LIN {X 0,Y 284.193,Z 792.338,A -85,B 0,C 180,E1 16435.65,E2 16435.65} C_VEL
LIN {X 0,Y 275.5,Z 813.457,A -85,B 0,C 180,E1 16443.138,E2 16443.138} C_VEL
LIN {X 0,Y 270.881,Z 827.883,A -85,B 0,C 180,E1 16450.476,E2 16450.476} C_VEL
LIN {X 0,Y 268.896,Z 838.261,A -85,B 0,C 180,E1 16458.673,E2 16458.673} C_VEL
LIN {X 0,Y 268.674,Z 843.154,A -85,B 0,C 180,E1 16466.783,E2 16466.783} C_VEL
LIN {X 0,Y 269.021,Z 843.604,A -85,B 0,C 180,E1 16470.002,E2 16470.002} C_VEL
LIN {X 0,Y 268.664,Z 840.876,A -85,B 0,C 180,E1 16478.074,E2 16478.074} C_VEL
LIN {X 0,Y 269.781,Z 832.628,A -85,B 0,C 180,E1 16486.243,E2 16486.243} C_VEL
LIN {X 0,Y 273.657,Z 818.429,A -85,B 0,C 180,E1 16494.453,E2 16494.453} C_VEL
LIN {X 0,Y 281.012,Z 798.576,A -85,B 0,C 180,E1 16502.079,E2 16502.079} C_VEL
LIN {X 0,Y 291.199,Z 773.618,A -85,B 0,C 180,E1 16508.743,E2 16508.743} C_VEL
LIN {X 0,Y 302.271,Z 746.073,A -85,B 0,C 180,E1 16513.948,E2 16513.948} C_VEL
LIN {X 0,Y 314,Z 714.004,A -85,B 0,C 180,E1 16518.227,E2 16518.227} C_VEL
LIN {X 0,Y 324.739,Z 678.752,A -85,B 0,C 180,E1 16521.486,E2 16521.486} C_VEL
LIN {X 0,Y 328.308,Z 663.259,A -85,B 0,C 180,E1 16522.637,E2 16522.637} C_VEL
LIN {X 0,Y 318.026,Z 633.867,A -85,B 0,C 180,E1 16527.518,E2 16527.518} C_VEL
LIN {X 0,Y 305.742,Z 608.81,A -85,B 0,C 180,E1 16532.476,E2 16532.476} C_VEL
LIN {X 0,Y 298.214,Z 601.214,A -85,B 0,C 180,E1 16535.1,E2 16535.1} C_VEL
LIN {X 0,Y 290.45,Z 594.981,A -85,B 0,C 180,E1 16537.97,E2 16537.97} C_VEL
LIN {X 0,Y 278.094,Z 576.688,A -85,B 0,C 180,E1 16543.729,E2 16543.729} C_VEL
LIN {X 0,Y 272.613,Z 569.407,A -85,B 0,C 180,E1 16546.675,E2 16546.675} C_VEL
LIN {X 0,Y 268.838,Z 563.675,A -85,B 0,C 180,E1 16549.01,E2 16549.01} C_VEL
LIN {X 0,Y 265.24,Z 558.237,A -85,B 0,C 180,E1 16551.479,E2 16551.479} C_VEL
LIN {X 0,Y 260.078,Z 551.896,A -85,B 0,C 180,E1 16555.502,E2 16555.502} C_VEL
LIN {X 0,Y 259.824,Z 549.53,A -85,B 0,C 180,E1 16556.227,E2 16556.227} C_VEL
LIN {X 0,Y 260.166,Z 549.53,A -85,B 0,C 180,E1 16559.972,E2 16559.972} C_VEL
LIN {X 0,Y 259.366,Z 549.53,A -85,B 0,C 180,E1 16568.461,E2 16568.461} C_VEL
LIN {X 0,Y 258.757,Z 549.53,A -85,B 0,C 180,E1 16576.92,E2 16576.92} C_VEL
LIN {X 0,Y 258.263,Z 549.53,A -85,B 0,C 180,E1 16584.106,E2 16584.106} C_VEL
LIN {X 0,Y 257.894,Z 549.53,A -85,B 0,C 180,E1 16591.736,E2 16591.736} C_VEL
LIN {X 0,Y 257.813,Z 549.77,A -85,B 0,C 180,E1 16595.549,E2 16595.549} C_VEL
LIN {X 0,Y 259.44,Z 554.315,A -85,B 0,C 180,E1 16597.326,E2 16597.326} C_VEL
LIN {X 0,Y 263.605,Z 557.866,A -85,B 0,C 180,E1 16600.498,E2 16600.498} C_VEL
LIN {X 0,Y 267.187,Z 563.441,A -85,B 0,C 180,E1 16603.061,E2 16603.061} C_VEL
LIN {X 0,Y 269.471,Z 566.342,A -85,B 0,C 180,E1 16604.516,E2 16604.516} C_VEL
LIN {X 0,Y 279.761,Z 580.464,A -85,B 0,C 180,E1 16610.268,E2 16610.268} C_VEL
LIN {X 0,Y 291.304,Z 599.056,A -85,B 0,C 180,E1 16616.073,E2 16616.073} C_VEL
LIN {X 0,Y 302.413,Z 621.809,A -85,B 0,C 180,E1 16621.67,E2 16621.67} C_VEL
LIN {X 0,Y 310.963,Z 646.908,A -85,B 0,C 180,E1 16626.849,E2 16626.849} C_VEL
LIN {X 0,Y 313.377,Z 660.612,A -85,B 0,C 180,E1 16629.324,E2 16629.324} C_VEL
LIN {X 0,Y 302.378,Z 694.403,A -85,B 0,C 180,E1 16633.136,E2 16633.136} C_VEL
LIN {X 0,Y 290.875,Z 723.87,A -85,B 0,C 180,E1 16638.021,E2 16638.021} C_VEL
LIN {X 0,Y 280.218,Z 748.211,A -85,B 0,C 180,E1 16643.815,E2 16643.815} C_VEL
LIN {X 0,Y 271.445,Z 767.751,A -85,B 0,C 180,E1 16650.553,E2 16650.553} C_VEL
LIN {X 0,Y 265.654,Z 781.533,A -85,B 0,C 180,E1 16657.597,E2 16657.597} C_VEL
LIN {X 0,Y 262.351,Z 790.678,A -85,B 0,C 180,E1 16664.998,E2 16664.998} C_VEL
LIN {X 0,Y 260.523,Z 795.27,A -85,B 0,C 180,E1 16672.171,E2 16672.171} C_VEL
LIN {X 0,Y 260.569,Z 795.838,A -85,B 0,C 180,E1 16679.773,E2 16679.773} C_VEL
LIN {X 0,Y 262.859,Z 791.758,A -85,B 0,C 180,E1 16687.666,E2 16687.666} C_VEL
LIN {X 0,Y 267.17,Z 782.441,A -85,B 0,C 180,E1 16695.737,E2 16695.737} C_VEL
LIN {X 0,Y 274.41,Z 768.233,A -85,B 0,C 180,E1 16703.143,E2 16703.143} C_VEL
LIN {X 0,Y 284.656,Z 748.679,A -85,B 0,C 180,E1 16709.894,E2 16709.894} C_VEL
LIN {X 0,Y 297.561,Z 722.75,A -85,B 0,C 180,E1 16715.894,E2 16715.894} C_VEL
LIN {X 0,Y 310.18,Z 693.863,A -85,B 0,C 180,E1 16720.466,E2 16720.466} C_VEL
LIN {X 0,Y 320.732,Z 664.253,A -85,B 0,C 180,E1 16723.806,E2 16723.806} C_VEL
LIN {X 0,Y 317.188,Z 642.293,A -85,B 0,C 180,E1 16728.708,E2 16728.708} C_VEL
LIN {X 0,Y 312.027,Z 624.584,A -85,B 0,C 180,E1 16733.778,E2 16733.778} C_VEL
LIN {X 0,Y 307.138,Z 612.298,A -85,B 0,C 180,E1 16738.842,E2 16738.842} C_VEL
LIN {X 0,Y 304.838,Z 607,A -85,B 0,C 180,E1 16741.993,E2 16741.993} C_VEL
LIN {X 0,Y 303.417,Z 603.216,A -85,B 0,C 180,E1 16744.94,E2 16744.94} C_VEL
LIN {X 0,Y 303.196,Z 603.27,A -85,B 0,C 180,E1 16754.063,E2 16754.063} C_VEL
LIN {X 0,Y 307.12,Z 611.288,A -85,B 0,C 180,E1 16760.137,E2 16760.137} C_VEL
LIN {X 0,Y 312.817,Z 623.081,A -85,B 0,C 180,E1 16765.242,E2 16765.242} C_VEL
LIN {X 0,Y 320.158,Z 641.035,A -85,B 0,C 180,E1 16770.477,E2 16770.477} C_VEL
LIN {X 0,Y 326.227,Z 663.874,A -85,B 0,C 180,E1 16775.218,E2 16775.218} C_VEL
LIN {X 0,Y 326.696,Z 668.857,A -85,B 0,C 180,E1 16775.992,E2 16775.992} C_VEL
LIN {X 0,Y 314.613,Z 705.853,A -85,B 0,C 180,E1 16779.162,E2 16779.162} C_VEL
LIN {X 0,Y 301.662,Z 738.296,A -85,B 0,C 180,E1 16783.245,E2 16783.245} C_VEL
LIN {X 0,Y 288.39,Z 767.968,A -85,B 0,C 180,E1 16788.618,E2 16788.618} C_VEL
LIN {X 0,Y 276.658,Z 793.34,A -85,B 0,C 180,E1 16795.194,E2 16795.194} C_VEL
LIN {X 0,Y 268.25,Z 812.802,A -85,B 0,C 180,E1 16802.351,E2 16802.351} C_VEL
LIN {X 0,Y 263.207,Z 827.19,A -85,B 0,C 180,E1 16809.882,E2 16809.882} C_VEL
LIN {X 0,Y 261.039,Z 837.525,A -85,B 0,C 180,E1 16818.285,E2 16818.285} C_VEL
LIN {X 0,Y 260.727,Z 841.111,A -85,B 0,C 180,E1 16823.355,E2 16823.355} C_VEL
LIN {X 0,Y 261.165,Z 842.891,A -85,B 0,C 180,E1 16830.002,E2 16830.002} C_VEL
LIN {X 0,Y 260.794,Z 840.13,A -85,B 0,C 180,E1 16838.32,E2 16838.32} C_VEL
LIN {X 0,Y 262.022,Z 831.837,A -85,B 0,C 180,E1 16846.738,E2 16846.738} C_VEL
LIN {X 0,Y 266.065,Z 817.867,A -85,B 0,C 180,E1 16855.034,E2 16855.034} C_VEL
LIN {X 0,Y 273.995,Z 797.737,A -85,B 0,C 180,E1 16862.95,E2 16862.95} C_VEL
LIN {X 0,Y 284.346,Z 773.493,A -85,B 0,C 180,E1 16869.559,E2 16869.559} C_VEL
LIN {X 0,Y 296.568,Z 744.344,A -85,B 0,C 180,E1 16875.119,E2 16875.119} C_VEL
LIN {X 0,Y 308.448,Z 712.855,A -85,B 0,C 180,E1 16879.318,E2 16879.318} C_VEL
LIN {X 0,Y 319.459,Z 677.531,A -85,B 0,C 180,E1 16882.577,E2 16882.577} C_VEL
LIN {X 0,Y 322.17,Z 666.238,A -85,B 0,C 180,E1 16883.423,E2 16883.423} C_VEL
LIN {X 0,Y 312.698,Z 638.024,A -85,B 0,C 180,E1 16888.326,E2 16888.326} C_VEL
LIN {X 0,Y 299.747,Z 610.961,A -85,B 0,C 180,E1 16893.944,E2 16893.944} C_VEL
LIN {X 0,Y 290.45,Z 594.981,A -85,B 0,C 180,E1 16897.97,E2 16897.97} C_VEL
LIN {X 0,Y 283.188,Z 588.984,A -85,B 0,C 180,E1 16900.923,E2 16900.923} C_VEL
LIN {X 0,Y 276.107,Z 584.174,A -85,B 0,C 180,E1 16904.09,E2 16904.09} C_VEL
LIN {X 0,Y 266.368,Z 570.629,A -85,B 0,C 180,E1 16909.817,E2 16909.817} C_VEL
LIN {X 0,Y 261.97,Z 564.047,A -85,B 0,C 180,E1 16913.015,E2 16913.015} C_VEL
LIN {X 0,Y 258.168,Z 558.953,A -85,B 0,C 180,E1 16916.203,E2 16916.203} C_VEL
LIN {X 0,Y 257.075,Z 556.909,A -85,B 0,C 180,E1 16917.287,E2 16917.287} C_VEL
LIN {X 0,Y 252.211,Z 551.414,A -85,B 0,C 180,E1 16922.757,E2 16922.757} C_VEL
LIN {X 0,Y 251.964,Z 549.53,A -85,B 0,C 180,E1 16923.404,E2 16923.404} C_VEL
LIN {X 0,Y 251.321,Z 549.53,A -85,B 0,C 180,E1 16930.346,E2 16930.346} C_VEL
LIN {X 0,Y 250.754,Z 549.53,A -85,B 0,C 180,E1 16937.477,E2 16937.477} C_VEL
LIN {X 0,Y 250.188,Z 549.53,A -85,B 0,C 180,E1 16945.207,E2 16945.207} C_VEL
LIN {X 0,Y 250.136,Z 550.202,A -85,B 0,C 180,E1 16947.393,E2 16947.393} C_VEL
LIN {X 0,Y 252.27,Z 555.117,A -85,B 0,C 180,E1 16951.01,E2 16951.01} C_VEL
LIN {X 0,Y 256.029,Z 558.069,A -85,B 0,C 180,E1 16955.039,E2 16955.039} C_VEL
LIN {X 0,Y 259.954,Z 563.878,A -85,B 0,C 180,E1 16958.662,E2 16958.662} C_VEL
LIN {X 0,Y 262.029,Z 566.363,A -85,B 0,C 180,E1 16960.268,E2 16960.268} C_VEL
LIN {X 0,Y 267.595,Z 574.233,A -85,B 0,C 180,E1 16964.204,E2 16964.204} C_VEL
LIN {X 0,Y 277.055,Z 587.648,A -85,B 0,C 180,E1 16969.829,E2 16969.829} C_VEL
LIN {X 0,Y 288.761,Z 607.478,A -85,B 0,C 180,E1 16976.143,E2 16976.143} C_VEL
LIN {X 0,Y 299.448,Z 631.987,A -85,B 0,C 180,E1 16982.154,E2 16982.154} C_VEL
LIN {X 0,Y 306.574,Z 656.821,A -85,B 0,C 180,E1 16987.324,E2 16987.324} C_VEL
LIN {X 0,Y 307.165,Z 663.632,A -85,B 0,C 180,E1 16988.511,E2 16988.511} C_VEL
LIN {X 0,Y 295.395,Z 697.825,A -85,B 0,C 180,E1 16992.533,E2 16992.533} C_VEL
LIN {X 0,Y 283.759,Z 726.213,A -85,B 0,C 180,E1 16997.43,E2 16997.43} C_VEL
LIN {X 0,Y 272.941,Z 749.863,A -85,B 0,C 180,E1 17003.266,E2 17003.266} C_VEL
LIN {X 0,Y 263.46,Z 770.089,A -85,B 0,C 180,E1 17010.57,E2 17010.57} C_VEL
LIN {X 0,Y 257.246,Z 784.193,A -85,B 0,C 180,E1 17018.429,E2 17018.429} C_VEL
LIN {X 0,Y 254.331,Z 792.082,A -85,B 0,C 180,E1 17025.483,E2 17025.483} C_VEL
LIN {X 0,Y 252.85,Z 795.586,A -85,B 0,C 180,E1 17030.98,E2 17030.98} C_VEL
LIN {X 0,Y 252.539,Z 796.787,A -85,B 0,C 180,E1 17038.554,E2 17038.554} C_VEL
LIN {X 0,Y 254.501,Z 793.76,A -85,B 0,C 180,E1 17046.362,E2 17046.362} C_VEL
LIN {X 0,Y 258.418,Z 785.884,A -85,B 0,C 180,E1 17054.482,E2 17054.482} C_VEL
LIN {X 0,Y 265.794,Z 772.126,A -85,B 0,C 180,E1 17062.635,E2 17062.635} C_VEL
LIN {X 0,Y 276.891,Z 752.114,A -85,B 0,C 180,E1 17070.101,E2 17070.101} C_VEL
LIN {X 0,Y 289.443,Z 728.439,A -85,B 0,C 180,E1 17076.006,E2 17076.006} C_VEL
LIN {X 0,Y 303.208,Z 699.093,A -85,B 0,C 180,E1 17081.007,E2 17081.007} C_VEL
LIN {X 0,Y 315.291,Z 668.078,A -85,B 0,C 180,E1 17084.608,E2 17084.608} C_VEL
LIN {X 0,Y 312.719,Z 648.093,A -85,B 0,C 180,E1 17089.249,E2 17089.249} C_VEL
LIN {X 0,Y 308.354,Z 630.717,A -85,B 0,C 180,E1 17094.408,E2 17094.408} C_VEL
LIN {X 0,Y 303.555,Z 616.33,A -85,B 0,C 180,E1 17100.645,E2 17100.645} C_VEL
LIN {X 0,Y 301.429,Z 610.831,A -85,B 0,C 180,E1 17104.973,E2 17104.973} C_VEL
LIN {X 0,Y 301.329,Z 610.961,A -85,B 0,C 180,E1 17114.166,E2 17114.166} C_VEL
LIN {X 0,Y 304.871,Z 619.297,A -85,B 0,C 180,E1 17120.122,E2 17120.122} C_VEL
LIN {X 0,Y 309.376,Z 629.152,A -85,B 0,C 180,E1 17124.513,E2 17124.513} C_VEL
LIN {X 0,Y 315.779,Z 646.279,A -85,B 0,C 180,E1 17129.742,E2 17129.742} C_VEL
LIN {X 0,Y 321.433,Z 670.42,A -85,B 0,C 180,E1 17134.918,E2 17134.918} C_VEL
LIN {X 0,Y 308.73,Z 707.743,A -85,B 0,C 180,E1 17138.243,E2 17138.243} C_VEL
LIN {X 0,Y 295.176,Z 740.016,A -85,B 0,C 180,E1 17142.435,E2 17142.435} C_VEL
LIN {X 0,Y 281.424,Z 769.211,A -85,B 0,C 180,E1 17147.916,E2 17147.916} C_VEL
LIN {X 0,Y 269.687,Z 793.231,A -85,B 0,C 180,E1 17154.356,E2 17154.356} C_VEL
LIN {X 0,Y 260.17,Z 813.986,A -85,B 0,C 180,E1 17162.357,E2 17162.357} C_VEL
LIN {X 0,Y 254.985,Z 828.322,A -85,B 0,C 180,E1 17170.515,E2 17170.515} C_VEL
LIN {X 0,Y 253.178,Z 836.864,A -85,B 0,C 180,E1 17177.962,E2 17177.962} C_VEL
LIN {X 0,Y 252.862,Z 840.419,A -85,B 0,C 180,E1 17183.148,E2 17183.148} C_VEL
LIN {X 0,Y 253.295,Z 842.177,A -85,B 0,C 180,E1 17190.003,E2 17190.003} C_VEL
LIN {X 0,Y 252.915,Z 839.376,A -85,B 0,C 180,E1 17198.581,E2 17198.581} C_VEL
LIN {X 0,Y 254.265,Z 831.021,A -85,B 0,C 180,E1 17207.265,E2 17207.265} C_VEL
LIN {X 0,Y 258.804,Z 816.51,A -85,B 0,C 180,E1 17216.021,E2 17216.021} C_VEL
LIN {X 0,Y 267.07,Z 796.721,A -85,B 0,C 180,E1 17223.918,E2 17223.918} C_VEL
LIN {X 0,Y 278.031,Z 772.344,A -85,B 0,C 180,E1 17230.643,E2 17230.643} C_VEL
LIN {X 0,Y 290.452,Z 743.771,A -85,B 0,C 180,E1 17236.152,E2 17236.152} C_VEL
LIN {X 0,Y 303.148,Z 711.203,A -85,B 0,C 180,E1 17240.498,E2 17240.498} C_VEL
LIN {X 0,Y 314.124,Z 677.015,A -85,B 0,C 180,E1 17243.641,E2 17243.641} C_VEL
LIN {X 0,Y 316.065,Z 669.09,A -85,B 0,C 180,E1 17244.26,E2 17244.26} C_VEL
LIN {X 0,Y 307.001,Z 641.23,A -85,B 0,C 180,E1 17249.319,E2 17249.319} C_VEL
LIN {X 0,Y 293.601,Z 612.659,A -85,B 0,C 180,E1 17255.6,E2 17255.6} C_VEL
LIN {X 0,Y 279.909,Z 589.895,A -85,B 0,C 180,E1 17262.122,E2 17262.122} C_VEL
LIN {X 0,Y 276.107,Z 584.174,A -85,B 0,C 180,E1 17264.09,E2 17264.09} C_VEL
LIN {X 0,Y 263.605,Z 577.022,A -85,B 0,C 180,E1 17270.887,E2 17270.887} C_VEL
LIN {X 0,Y 260.029,Z 571.373,A -85,B 0,C 180,E1 17273.622,E2 17273.622} C_VEL
LIN {X 0,Y 256.155,Z 565.473,A -85,B 0,C 180,E1 17277.078,E2 17277.078} C_VEL
LIN {X 0,Y 250.678,Z 558.6,A -85,B 0,C 180,E1 17283.422,E2 17283.422} C_VEL
LIN {X 0,Y 250.175,Z 557.261,A -85,B 0,C 180,E1 17284.294,E2 17284.294} C_VEL
LIN {X 0,Y 245.952,Z 555.911,A -85,B 0,C 180,E1 17298.515,E2 17298.515} C_VEL
LIN {X 0,Y 248.805,Z 558.137,A -85,B 0,C 180,E1 17307.018,E2 17307.018} C_VEL
LIN {X 0,Y 251.434,Z 563.222,A -85,B 0,C 180,E1 17311.324,E2 17311.324} C_VEL
LIN {X 0,Y 254.418,Z 565.787,A -85,B 0,C 180,E1 17314.584,E2 17314.584} C_VEL
LIN {X 0,Y 259.015,Z 571.897,A -85,B 0,C 180,E1 17318.829,E2 17318.829} C_VEL
LIN {X 0,Y 265.964,Z 582.469,A -85,B 0,C 180,E1 17324.121,E2 17324.121} C_VEL
LIN {X 0,Y 276.085,Z 597.607,A -85,B 0,C 180,E1 17330.481,E2 17330.481} C_VEL
LIN {X 0,Y 286.656,Z 617.794,A -85,B 0,C 180,E1 17336.688,E2 17336.688} C_VEL
LIN {X 0,Y 295.33,Z 639.991,A -85,B 0,C 180,E1 17342.18,E2 17342.18} C_VEL
LIN {X 0,Y 301.105,Z 663.201,A -85,B 0,C 180,E1 17347.143,E2 17347.143} C_VEL
LIN {X 0,Y 300.365,Z 668.459,A -85,B 0,C 180,E1 17347.862,E2 17347.862} C_VEL
LIN {X 0,Y 288.456,Z 701.169,A -85,B 0,C 180,E1 17351.902,E2 17351.902} C_VEL
LIN {X 0,Y 276.32,Z 729.352,A -85,B 0,C 180,E1 17356.978,E2 17356.978} C_VEL
LIN {X 0,Y 264.507,Z 753.919,A -85,B 0,C 180,E1 17363.446,E2 17363.446} C_VEL
LIN {X 0,Y 255.21,Z 772.77,A -85,B 0,C 180,E1 17370.844,E2 17370.844} C_VEL
LIN {X 0,Y 249.197,Z 785.882,A -85,B 0,C 180,E1 17378.705,E2 17378.705} C_VEL
LIN {X 0,Y 246.3,Z 793.365,A -85,B 0,C 180,E1 17386.001,E2 17386.001} C_VEL
LIN {X 0,Y 244.696,Z 796.81,A -85,B 0,C 180,E1 17392.437,E2 17392.437} C_VEL
LIN {X 0,Y 244.915,Z 797.207,A -85,B 0,C 180,E1 17400.472,E2 17400.472} C_VEL
LIN {X 0,Y 247.119,Z 793.967,A -85,B 0,C 180,E1 17407.633,E2 17407.633} C_VEL
LIN {X 0,Y 251.602,Z 785.533,A -85,B 0,C 180,E1 17416.027,E2 17416.027} C_VEL
LIN {X 0,Y 259.945,Z 771.041,A -85,B 0,C 180,E1 17424.358,E2 17424.358} C_VEL
LIN {X 0,Y 271.372,Z 751.572,A -85,B 0,C 180,E1 17431.548,E2 17431.548} C_VEL
LIN {X 0,Y 285.396,Z 726.339,A -85,B 0,C 180,E1 17437.73,E2 17437.73} C_VEL
LIN {X 0,Y 299.543,Z 696.829,A -85,B 0,C 180,E1 17442.583,E2 17442.583} C_VEL
LIN {X 0,Y 309.854,Z 671.078,A -85,B 0,C 180,E1 17445.618,E2 17445.618} C_VEL
LIN {X 0,Y 307.729,Z 651.292,A -85,B 0,C 180,E1 17450.5,E2 17450.5} C_VEL
LIN {X 0,Y 304.006,Z 634.947,A -85,B 0,C 180,E1 17455.755,E2 17455.755} C_VEL
LIN {X 0,Y 300.598,Z 623.227,A -85,B 0,C 180,E1 17461.279,E2 17461.279} C_VEL
LIN {X 0,Y 299.106,Z 618.349,A -85,B 0,C 180,E1 17465.088,E2 17465.088} C_VEL
LIN {X 0,Y 299.232,Z 618.571,A -85,B 0,C 180,E1 17474.268,E2 17474.268} C_VEL
LIN {X 0,Y 301.996,Z 625.941,A -85,B 0,C 180,E1 17479.501,E2 17479.501} C_VEL
LIN {X 0,Y 306.726,Z 637.711,A -85,B 0,C 180,E1 17484.739,E2 17484.739} C_VEL
LIN {X 0,Y 312.278,Z 654.88,A -85,B 0,C 180,E1 17489.846,E2 17489.846} C_VEL
LIN {X 0,Y 315.852,Z 673.028,A -85,B 0,C 180,E1 17493.858,E2 17493.858} C_VEL
LIN {X 0,Y 303.712,Z 707.731,A -85,B 0,C 180,E1 17497.076,E2 17497.076} C_VEL
LIN {X 0,Y 289.87,Z 739.318,A -85,B 0,C 180,E1 17501.197,E2 17501.197} C_VEL
LIN {X 0,Y 275.375,Z 768.702,A -85,B 0,C 180,E1 17506.769,E2 17506.769} C_VEL
LIN {X 0,Y 262.649,Z 793.457,A -85,B 0,C 180,E1 17513.575,E2 17513.575} C_VEL
LIN {X 0,Y 252.949,Z 813.356,A -85,B 0,C 180,E1 17521.497,E2 17521.497} C_VEL
LIN {X 0,Y 247.389,Z 827.47,A -85,B 0,C 180,E1 17529.755,E2 17529.755} C_VEL
LIN {X 0,Y 245.333,Z 836.17,A -85,B 0,C 180,E1 17537.571,E2 17537.571} C_VEL
LIN {X 0,Y 244.978,Z 839.727,A -85,B 0,C 180,E1 17542.926,E2 17542.926} C_VEL
LIN {X 0,Y 245.437,Z 841.462,A -85,B 0,C 180,E1 17550.003,E2 17550.003} C_VEL
LIN {X 0,Y 244.989,Z 839.575,A -85,B 0,C 180,E1 17557.079,E2 17557.079} C_VEL
LIN {X 0,Y 246.047,Z 832.29,A -85,B 0,C 180,E1 17566.024,E2 17566.024} C_VEL
LIN {X 0,Y 250.071,Z 819.131,A -85,B 0,C 180,E1 17574.989,E2 17574.989} C_VEL
LIN {X 0,Y 258.051,Z 800.5,A -85,B 0,C 180,E1 17583.248,E2 17583.248} C_VEL
LIN {X 0,Y 269.613,Z 775.845,A -85,B 0,C 180,E1 17590.679,E2 17590.679} C_VEL
LIN {X 0,Y 283.362,Z 745.72,A -85,B 0,C 180,E1 17596.804,E2 17596.804} C_VEL
LIN {X 0,Y 296.361,Z 713.854,A -85,B 0,C 180,E1 17601.235,E2 17601.235} C_VEL
LIN {X 0,Y 307.832,Z 679.957,A -85,B 0,C 180,E1 17604.476,E2 17604.476} C_VEL
LIN {X 0,Y 310.048,Z 672.07,A -85,B 0,C 180,E1 17605.1,E2 17605.1} C_VEL
LIN {X 0,Y 301.352,Z 644.503,A -85,B 0,C 180,E1 17610.344,E2 17610.344} C_VEL
LIN {X 0,Y 288.95,Z 617.37,A -85,B 0,C 180,E1 17616.614,E2 17616.614} C_VEL
LIN {X 0,Y 276.709,Z 596.132,A -85,B 0,C 180,E1 17622.932,E2 17622.932} C_VEL
LIN {X 0,Y 267.303,Z 582.249,A -85,B 0,C 180,E1 17628.415,E2 17628.415} C_VEL
LIN {X 0,Y 263.701,Z 577.137,A -85,B 0,C 180,E1 17630.821,E2 17630.821} C_VEL
LIN {X 0,Y 263.605,Z 577.022,A -85,B 0,C 180,E1 17630.887,E2 17630.887} C_VEL
LIN {X 0,Y 258.528,Z 573.47,A -85,B 0,C 180,E1 17634.46,E2 17634.46} C_VEL
LIN {X 0,Y 253.87,Z 572.117,A -85,B 0,C 180,E1 17638.241,E2 17638.241} C_VEL
LIN {X 0,Y 249.239,Z 566.032,A -85,B 0,C 180,E1 17643.961,E2 17643.961} C_VEL
LIN {X 0,Y 246.48,Z 564.258,A -85,B 0,C 180,E1 17648.858,E2 17648.858} C_VEL
LIN {X 0,Y 245.229,Z 564.074,A -85,B 0,C 180,E1 17660.652,E2 17660.652} C_VEL
LIN {X 0,Y 247.522,Z 565.974,A -85,B 0,C 180,E1 17666.68,E2 17666.68} C_VEL
LIN {X 0,Y 250.608,Z 571.369,A -85,B 0,C 180,E1 17671.649,E2 17671.649} C_VEL
LIN {X 0,Y 252.895,Z 573.689,A -85,B 0,C 180,E1 17674.265,E2 17674.265} C_VEL
LIN {X 0,Y 258.311,Z 581.617,A -85,B 0,C 180,E1 17679.445,E2 17679.445} C_VEL
LIN {X 0,Y 266.227,Z 593.425,A -85,B 0,C 180,E1 17685.525,E2 17685.525} C_VEL
LIN {X 0,Y 276.436,Z 611.135,A -85,B 0,C 180,E1 17692.279,E2 17692.279} C_VEL
LIN {X 0,Y 286.105,Z 632.907,A -85,B 0,C 180,E1 17698.565,E2 17698.565} C_VEL
LIN {X 0,Y 293.42,Z 657.173,A -85,B 0,C 180,E1 17704.33,E2 17704.33} C_VEL
LIN {X 0,Y 295.03,Z 668.901,A -85,B 0,C 180,E1 17706.743,E2 17706.743} C_VEL
LIN {X 0,Y 282.873,Z 701.133,A -85,B 0,C 180,E1 17710.724,E2 17710.724} C_VEL
LIN {X 0,Y 270.26,Z 729.472,A -85,B 0,C 180,E1 17715.858,E2 17715.858} C_VEL
LIN {X 0,Y 258.167,Z 753.697,A -85,B 0,C 180,E1 17722.254,E2 17722.254} C_VEL
LIN {X 0,Y 248.068,Z 773.182,A -85,B 0,C 180,E1 17729.997,E2 17729.997} C_VEL
LIN {X 0,Y 241.652,Z 786.389,A -85,B 0,C 180,E1 17738.074,E2 17738.074} C_VEL
LIN {X 0,Y 238.316,Z 794.447,A -85,B 0,C 180,E1 17746.308,E2 17746.308} C_VEL
LIN {X 0,Y 236.815,Z 797.543,A -85,B 0,C 180,E1 17752.475,E2 17752.475} C_VEL
LIN {X 0,Y 237.078,Z 797.948,A -85,B 0,C 180,E1 17760.608,E2 17760.608} C_VEL
LIN {X 0,Y 239.755,Z 794.032,A -85,B 0,C 180,E1 17769.002,E2 17769.002} C_VEL
LIN {X 0,Y 244.952,Z 785.044,A -85,B 0,C 180,E1 17777.664,E2 17777.664} C_VEL
LIN {X 0,Y 253.16,Z 771.818,A -85,B 0,C 180,E1 17785.321,E2 17785.321} C_VEL
LIN {X 0,Y 264.473,Z 753.677,A -85,B 0,C 180,E1 17792.245,E2 17792.245} C_VEL
LIN {X 0,Y 278.522,Z 729.668,A -85,B 0,C 180,E1 17798.389,E2 17798.389} C_VEL
LIN {X 0,Y 293.456,Z 700.487,A -85,B 0,C 180,E1 17803.416,E2 17803.416} C_VEL
LIN {X 0,Y 304.505,Z 673.757,A -85,B 0,C 180,E1 17806.721,E2 17806.721} C_VEL
LIN {X 0,Y 302.872,Z 654.631,A -85,B 0,C 180,E1 17811.755,E2 17811.755} C_VEL
LIN {X 0,Y 299.882,Z 639.209,A -85,B 0,C 180,E1 17817.14,E2 17817.14} C_VEL
LIN {X 0,Y 297.776,Z 630.603,A -85,B 0,C 180,E1 17821.476,E2 17821.476} C_VEL
LIN {X 0,Y 296.312,Z 625.726,A -85,B 0,C 180,E1 17825.869,E2 17825.869} C_VEL
LIN {X 0,Y 296.029,Z 625.451,A -85,B 0,C 180,E1 17831.787,E2 17831.787} C_VEL
LIN {X 0,Y 297.299,Z 628.815,A -85,B 0,C 180,E1 17836.015,E2 17836.015} C_VEL
LIN {X 0,Y 299.608,Z 634.412,A -85,B 0,C 180,E1 17839.896,E2 17839.896} C_VEL
LIN {X 0,Y 303.884,Z 646.379,A -85,B 0,C 180,E1 17845.027,E2 17845.027} C_VEL
LIN {X 0,Y 308.218,Z 662.752,A -85,B 0,C 180,E1 17849.799,E2 17849.799} C_VEL
LIN {X 0,Y 310.418,Z 677.442,A -85,B 0,C 180,E1 17853.072,E2 17853.072} C_VEL
LIN {X 0,Y 296.051,Z 714.4,A -85,B 0,C 180,E1 17856.605,E2 17856.605} C_VEL
LIN {X 0,Y 280.848,Z 746.554,A -85,B 0,C 180,E1 17861.22,E2 17861.22} C_VEL
LIN {X 0,Y 266.041,Z 774.562,A -85,B 0,C 180,E1 17867.109,E2 17867.109} C_VEL
LIN {X 0,Y 253.04,Z 798.447,A -85,B 0,C 180,E1 17874.451,E2 17874.451} C_VEL
LIN {X 0,Y 244.09,Z 816.194,A -85,B 0,C 180,E1 17882.379,E2 17882.379} C_VEL
LIN {X 0,Y 238.761,Z 829.932,A -85,B 0,C 180,E1 17891.581,E2 17891.581} C_VEL
LIN {X 0,Y 237.185,Z 837.736,A -85,B 0,C 180,E1 17900.303,E2 17900.303} C_VEL
LIN {X 0,Y 237.118,Z 840.336,A -85,B 0,C 180,E1 17906.354,E2 17906.354} C_VEL
LIN {X 0,Y 237.556,Z 840.745,A -85,B 0,C 180,E1 17910.003,E2 17910.003} C_VEL
LIN {X 0,Y 237.097,Z 838.828,A -85,B 0,C 180,E1 17917.316,E2 17917.316} C_VEL
LIN {X 0,Y 237.817,Z 833.451,A -85,B 0,C 180,E1 17924.706,E2 17924.706} C_VEL
LIN {X 0,Y 241.434,Z 821.463,A -85,B 0,C 180,E1 17933.962,E2 17933.962} C_VEL
LIN {X 0,Y 249.503,Z 802.915,A -85,B 0,C 180,E1 17942.982,E2 17942.982} C_VEL
LIN {X 0,Y 260.434,Z 780.624,A -85,B 0,C 180,E1 17950.284,E2 17950.284} C_VEL
LIN {X 0,Y 273.434,Z 753.684,A -85,B 0,C 180,E1 17956.391,E2 17956.391} C_VEL
LIN {X 0,Y 286.925,Z 723.017,A -85,B 0,C 180,E1 17961.18,E2 17961.18} C_VEL
LIN {X 0,Y 299.632,Z 688.611,A -85,B 0,C 180,E1 17964.859,E2 17964.859} C_VEL
LIN {X 0,Y 303.781,Z 674.278,A -85,B 0,C 180,E1 17966.093,E2 17966.093} C_VEL
LIN {X 0,Y 295.731,Z 647.769,A -85,B 0,C 180,E1 17971.4,E2 17971.4} C_VEL
LIN {X 0,Y 283.731,Z 620.569,A -85,B 0,C 180,E1 17978.018,E2 17978.018} C_VEL
LIN {X 0,Y 271.318,Z 598.53,A -85,B 0,C 180,E1 17985.023,E2 17985.023} C_VEL
LIN {X 0,Y 261.6,Z 584.268,A -85,B 0,C 180,E1 17991.421,E2 17991.421} C_VEL
LIN {X 0,Y 257.786,Z 578.387,A -85,B 0,C 180,E1 17994.504,E2 17994.504} C_VEL
LIN {X 0,Y 253.87,Z 572.117,A -85,B 0,C 180,E1 17998.241,E2 17998.241} C_VEL
LIN {X 0,Y 246.891,Z 572.604,A -85,B 0,C 180,E1 18006.074,E2 18006.074} C_VEL
LIN {X 0,Y 243.851,Z 571.575,A -85,B 0,C 180,E1 18018.681,E2 18018.681} C_VEL
LIN {X 0,Y 246.204,Z 573.681,A -85,B 0,C 180,E1 18026.264,E2 18026.264} C_VEL
LIN {X 0,Y 249.71,Z 579.475,A -85,B 0,C 180,E1 18032.075,E2 18032.075} C_VEL
LIN {X 0,Y 251.469,Z 581.932,A -85,B 0,C 180,E1 18034.19,E2 18034.19} C_VEL
LIN {X 0,Y 256.299,Z 589.375,A -85,B 0,C 180,E1 18039.194,E2 18039.194} C_VEL
LIN {X 0,Y 263.278,Z 600.304,A -85,B 0,C 180,E1 18044.96,E2 18044.96} C_VEL
LIN {X 0,Y 272.521,Z 617.101,A -85,B 0,C 180,E1 18051.573,E2 18051.573} C_VEL
LIN {X 0,Y 281.568,Z 638.937,A -85,B 0,C 180,E1 18058.09,E2 18058.09} C_VEL
LIN {X 0,Y 287.798,Z 661.779,A -85,B 0,C 180,E1 18063.723,E2 18063.723} C_VEL
LIN {X 0,Y 289.25,Z 670.824,A -85,B 0,C 180,E1 18065.74,E2 18065.74} C_VEL
LIN {X 0,Y 276.519,Z 703.305,A -85,B 0,C 180,E1 18069.847,E2 18069.847} C_VEL
LIN {X 0,Y 263.486,Z 731.305,A -85,B 0,C 180,E1 18075.063,E2 18075.063} C_VEL
LIN {X 0,Y 250.578,Z 755.872,A -85,B 0,C 180,E1 18081.837,E2 18081.837} C_VEL
LIN {X 0,Y 240.867,Z 773.783,A -85,B 0,C 180,E1 18089.204,E2 18089.204} C_VEL
LIN {X 0,Y 234.162,Z 786.883,A -85,B 0,C 180,E1 18097.402,E2 18097.402} C_VEL
LIN {X 0,Y 230.766,Z 794.553,A -85,B 0,C 180,E1 18105.16,E2 18105.16} C_VEL
LIN {X 0,Y 228.843,Z 798.52,A -85,B 0,C 180,E1 18113.303,E2 18113.303} C_VEL
LIN {X 0,Y 229.404,Z 798.483,A -85,B 0,C 180,E1 18121.748,E2 18121.748} C_VEL
LIN {X 0,Y 232.516,Z 794.09,A -85,B 0,C 180,E1 18130.462,E2 18130.462} C_VEL
LIN {X 0,Y 238.544,Z 784.589,A -85,B 0,C 180,E1 18139.382,E2 18139.382} C_VEL
LIN {X 0,Y 248.98,Z 768.922,A -85,B 0,C 180,E1 18148.045,E2 18148.045} C_VEL
LIN {X 0,Y 262.779,Z 747.75,A -85,B 0,C 180,E1 18155.398,E2 18155.398} C_VEL
LIN {X 0,Y 277.489,Z 722.861,A -85,B 0,C 180,E1 18161.145,E2 18161.145} C_VEL
LIN {X 0,Y 292.639,Z 693.139,A -85,B 0,C 180,E1 18165.759,E2 18165.759} C_VEL
LIN {X 0,Y 299.165,Z 678.17,A -85,B 0,C 180,E1 18167.491,E2 18167.491} C_VEL
LIN {X 0,Y 298.531,Z 661.383,A -85,B 0,C 180,E1 18172.036,E2 18172.036} C_VEL
LIN {X 0,Y 296.192,Z 645.285,A -85,B 0,C 180,E1 18177.835,E2 18177.835} C_VEL
LIN {X 0,Y 294.274,Z 636.295,A -85,B 0,C 180,E1 18182.963,E2 18182.963} C_VEL
LIN {X 0,Y 293.683,Z 633.203,A -85,B 0,C 180,E1 18185.922,E2 18185.922} C_VEL
LIN {X 0,Y 293.526,Z 633.236,A -85,B 0,C 180,E1 18192.379,E2 18192.379} C_VEL
LIN {X 0,Y 295.661,Z 638.531,A -85,B 0,C 180,E1 18197.854,E2 18197.854} C_VEL
LIN {X 0,Y 299.521,Z 650.799,A -85,B 0,C 180,E1 18203.789,E2 18203.789} C_VEL
LIN {X 0,Y 303.421,Z 666.839,A -85,B 0,C 180,E1 18208.822,E2 18208.822} C_VEL
LIN {X 0,Y 304.99,Z 680.919,A -85,B 0,C 180,E1 18212.085,E2 18212.085} C_VEL
LIN {X 0,Y 290.122,Z 716.775,A -85,B 0,C 180,E1 18215.643,E2 18215.643} C_VEL
LIN {X 0,Y 274.533,Z 748.099,A -85,B 0,C 180,E1 18220.288,E2 18220.288} C_VEL
LIN {X 0,Y 259.491,Z 775.135,A -85,B 0,C 180,E1 18226.154,E2 18226.154} C_VEL
LIN {X 0,Y 245.745,Z 799.017,A -85,B 0,C 180,E1 18233.773,E2 18233.773} C_VEL
LIN {X 0,Y 236.023,Z 817.211,A -85,B 0,C 180,E1 18242.388,E2 18242.388} C_VEL
LIN {X 0,Y 230.746,Z 830.378,A -85,B 0,C 180,E1 18251.945,E2 18251.945} C_VEL
LIN {X 0,Y 229.229,Z 837.605,A -85,B 0,C 180,E1 18261.027,E2 18261.027} C_VEL
LIN {X 0,Y 229.696,Z 840.03,A -85,B 0,C 180,E1 18270.003,E2 18270.003} C_VEL
LIN {X 0,Y 229.242,Z 837.39,A -85,B 0,C 180,E1 18278.994,E2 18278.994} C_VEL
LIN {X 0,Y 230.82,Z 829.669,A -85,B 0,C 180,E1 18288.065,E2 18288.065} C_VEL
LIN {X 0,Y 236.036,Z 815.704,A -85,B 0,C 180,E1 18297.616,E2 18297.616} C_VEL
LIN {X 0,Y 245.534,Z 796.136,A -85,B 0,C 180,E1 18306.249,E2 18306.249} C_VEL
LIN {X 0,Y 258.213,Z 771.614,A -85,B 0,C 180,E1 18313.528,E2 18313.528} C_VEL
LIN {X 0,Y 272.282,Z 742.859,A -85,B 0,C 180,E1 18319.342,E2 18319.342} C_VEL
LIN {X 0,Y 286.436,Z 709.973,A -85,B 0,C 180,E1 18323.858,E2 18323.858} C_VEL
LIN {X 0,Y 297.623,Z 676.883,A -85,B 0,C 180,E1 18327.056,E2 18327.056} C_VEL
LIN {X 0,Y 290.225,Z 651.415,A -85,B 0,C 180,E1 18332.381,E2 18332.381} C_VEL
LIN {X 0,Y 279.173,Z 625.523,A -85,B 0,C 180,E1 18338.994,E2 18338.994} C_VEL
LIN {X 0,Y 268.238,Z 605.105,A -85,B 0,C 180,E1 18345.765,E2 18345.765} C_VEL
LIN {X 0,Y 259.345,Z 591.235,A -85,B 0,C 180,E1 18352.102,E2 18352.102} C_VEL
LIN {X 0,Y 255.716,Z 585.561,A -85,B 0,C 180,E1 18355.18,E2 18355.18} C_VEL
LIN {X 0,Y 251.662,Z 579.273,A -85,B 0,C 180,E1 18359.327,E2 18359.327} C_VEL
LIN {X 0,Y 247.246,Z 572.715,A -85,B 0,C 180,E1 18365.485,E2 18365.485} C_VEL
LIN {X 0,Y 246.891,Z 572.604,A -85,B 0,C 180,E1 18366.074,E2 18366.074} C_VEL
LIN {X 0,Y 244.44,Z 575.773,A -85,B 0,C 180,E1 18370.058,E2 18370.058} C_VEL
LIN {X 0,Y 242.794,Z 579.171,A -85,B 0,C 180,E1 18374.102,E2 18374.102} C_VEL
LIN {X 0,Y 244.768,Z 581.34,A -85,B 0,C 180,E1 18385.87,E2 18385.87} C_VEL
LIN {X 0,Y 248.207,Z 587.224,A -85,B 0,C 180,E1 18391.991,E2 18391.991} C_VEL
LIN {X 0,Y 253.905,Z 596.536,A -85,B 0,C 180,E1 18398.664,E2 18398.664} C_VEL
LIN {X 0,Y 260.58,Z 607.872,A -85,B 0,C 180,E1 18404.684,E2 18404.684} C_VEL
LIN {X 0,Y 269.419,Z 625.179,A -85,B 0,C 180,E1 18411.581,E2 18411.581} C_VEL
LIN {X 0,Y 277.461,Z 646.684,A -85,B 0,C 180,E1 18418.09,E2 18418.09} C_VEL
LIN {X 0,Y 282.506,Z 668.397,A -85,B 0,C 180,E1 18423.553,E2 18423.553} C_VEL
LIN {X 0,Y 282.751,Z 674.949,A -85,B 0,C 180,E1 18424.934,E2 18424.934} C_VEL
LIN {X 0,Y 269.287,Z 707.594,A -85,B 0,C 180,E1 18429.281,E2 18429.281} C_VEL
LIN {X 0,Y 255.005,Z 736.267,A -85,B 0,C 180,E1 18434.993,E2 18434.993} C_VEL
LIN {X 0,Y 242.516,Z 758.93,A -85,B 0,C 180,E1 18441.709,E2 18441.709} C_VEL
LIN {X 0,Y 232,Z 777.469,A -85,B 0,C 180,E1 18449.997,E2 18449.997} C_VEL
LIN {X 0,Y 225.536,Z 789.708,A -85,B 0,C 180,E1 18458.655,E2 18458.655} C_VEL
LIN {X 0,Y 221.995,Z 797.201,A -85,B 0,C 180,E1 18468.036,E2 18468.036} C_VEL
LIN {X 0,Y 220.93,Z 799.735,A -85,B 0,C 180,E1 18477.482,E2 18477.482} C_VEL
LIN {X 0,Y 222.671,Z 798.021,A -85,B 0,C 180,E1 18485.662,E2 18485.662} C_VEL
LIN {X 0,Y 227.605,Z 790.916,A -85,B 0,C 180,E1 18495.61,E2 18495.61} C_VEL
LIN {X 0,Y 236.614,Z 777.966,A -85,B 0,C 180,E1 18505.019,E2 18505.019} C_VEL
LIN {X 0,Y 249.49,Z 759.761,A -85,B 0,C 180,E1 18513.104,E2 18513.104} C_VEL
LIN {X 0,Y 265.225,Z 735.936,A -85,B 0,C 180,E1 18519.884,E2 18519.884} C_VEL
LIN {X 0,Y 281.078,Z 708.206,A -85,B 0,C 180,E1 18525.088,E2 18525.088} C_VEL
LIN {X 0,Y 294.107,Z 680.619,A -85,B 0,C 180,E1 18528.734,E2 18528.734} C_VEL
LIN {X 0,Y 293.769,Z 663.593,A -85,B 0,C 180,E1 18533.759,E2 18533.759} C_VEL
LIN {X 0,Y 292.193,Z 649.743,A -85,B 0,C 180,E1 18539.285,E2 18539.285} C_VEL
LIN {X 0,Y 291.024,Z 641.998,A -85,B 0,C 180,E1 18544.363,E2 18544.363} C_VEL
LIN {X 0,Y 290.349,Z 640.11,A -85,B 0,C 180,E1 18549.092,E2 18549.092} C_VEL
LIN {X 0,Y 290.987,Z 641.426,A -85,B 0,C 180,E1 18553.517,E2 18553.517} C_VEL
LIN {X 0,Y 293.321,Z 648.541,A -85,B 0,C 180,E1 18559.291,E2 18559.291} C_VEL
LIN {X 0,Y 296.805,Z 661.598,A -85,B 0,C 180,E1 18564.938,E2 18564.938} C_VEL
LIN {X 0,Y 299.559,Z 678.829,A -85,B 0,C 180,E1 18569.868,E2 18569.868} C_VEL
LIN {X 0,Y 299.511,Z 684.485,A -85,B 0,C 180,E1 18571.078,E2 18571.078} C_VEL
LIN {X 0,Y 284.303,Z 719.233,A -85,B 0,C 180,E1 18574.648,E2 18574.648} C_VEL
LIN {X 0,Y 268.245,Z 749.825,A -85,B 0,C 180,E1 18579.334,E2 18579.334} C_VEL
LIN {X 0,Y 252.041,Z 777.395,A -85,B 0,C 180,E1 18585.588,E2 18585.588} C_VEL
LIN {X 0,Y 237.146,Z 801.81,A -85,B 0,C 180,E1 18593.968,E2 18593.968} C_VEL
LIN {X 0,Y 227.108,Z 819.988,A -85,B 0,C 180,E1 18603.58,E2 18603.58} C_VEL
LIN {X 0,Y 222.596,Z 831.21,A -85,B 0,C 180,E1 18612.803,E2 18612.803} C_VEL
LIN {X 0,Y 221.341,Z 837.666,A -85,B 0,C 180,E1 18622.166,E2 18622.166} C_VEL
LIN {X 0,Y 221.812,Z 839.31,A -85,B 0,C 180,E1 18630.003,E2 18630.003} C_VEL
LIN {X 0,Y 221.363,Z 836.623,A -85,B 0,C 180,E1 18639.317,E2 18639.317} C_VEL
LIN {X 0,Y 223.111,Z 828.856,A -85,B 0,C 180,E1 18648.697,E2 18648.697} C_VEL
LIN {X 0,Y 228.788,Z 814.764,A -85,B 0,C 180,E1 18658.57,E2 18658.57} C_VEL
LIN {X 0,Y 238.788,Z 795.262,A -85,B 0,C 180,E1 18667.351,E2 18667.351} C_VEL
LIN {X 0,Y 251.844,Z 771.067,A -85,B 0,C 180,E1 18674.653,E2 18674.653} C_VEL
LIN {X 0,Y 266.419,Z 742.46,A -85,B 0,C 180,E1 18680.513,E2 18680.513} C_VEL
LIN {X 0,Y 280.919,Z 709.936,A -85,B 0,C 180,E1 18685.009,E2 18685.009} C_VEL
LIN {X 0,Y 291.635,Z 679.947,A -85,B 0,C 180,E1 18687.949,E2 18687.949} C_VEL
LIN {X 0,Y 284.921,Z 655.597,A -85,B 0,C 180,E1 18693.293,E2 18693.293} C_VEL
LIN {X 0,Y 274.594,Z 630.204,A -85,B 0,C 180,E1 18700.072,E2 18700.072} C_VEL
LIN {X 0,Y 264.783,Z 611.283,A -85,B 0,C 180,E1 18706.624,E2 18706.624} C_VEL
LIN {X 0,Y 256.23,Z 597.05,A -85,B 0,C 180,E1 18713.315,E2 18713.315} C_VEL
LIN {X 0,Y 250.2,Z 586.98,A -85,B 0,C 180,E1 18719.539,E2 18719.539} C_VEL
LIN {X 0,Y 245.637,Z 580.36,A -85,B 0,C 180,E1 18726.273,E2 18726.273} C_VEL
LIN {X 0,Y 242.794,Z 579.171,A -85,B 0,C 180,E1 18734.102,E2 18734.102} C_VEL
LIN {X 0,Y 242.22,Z 581.725,A -85,B 0,C 180,E1 18737.143,E2 18737.143} C_VEL
LIN {X 0,Y 241.921,Z 587.604,A -85,B 0,C 180,E1 18741.644,E2 18741.644} C_VEL
LIN {X 0,Y 242.032,Z 587.766,A -85,B 0,C 180,E1 18742.164,E2 18742.164} C_VEL
LIN {X 0,Y 243.214,Z 589.297,A -85,B 0,C 180,E1 18745.702,E2 18745.702} C_VEL
LIN {X 0,Y 246.844,Z 595.094,A -85,B 0,C 180,E1 18752.28,E2 18752.28} C_VEL
LIN {X 0,Y 251.924,Z 604.852,A -85,B 0,C 180,E1 18758.8,E2 18758.8} C_VEL
LIN {X 0,Y 257.695,Z 615.341,A -85,B 0,C 180,E1 18764.404,E2 18764.404} C_VEL
LIN {X 0,Y 266.066,Z 633.006,A -85,B 0,C 180,E1 18771.592,E2 18771.592} C_VEL
LIN {X 0,Y 273.031,Z 654.269,A -85,B 0,C 180,E1 18778.091,E2 18778.091} C_VEL
LIN {X 0,Y 277.205,Z 676.314,A -85,B 0,C 180,E1 18783.766,E2 18783.766} C_VEL
LIN {X 0,Y 263.501,Z 708.565,A -85,B 0,C 180,E1 18788.143,E2 18788.143} C_VEL
LIN {X 0,Y 249.177,Z 736.353,A -85,B 0,C 180,E1 18793.732,E2 18793.732} C_VEL
LIN {X 0,Y 235.882,Z 759.45,A -85,B 0,C 180,E1 18800.653,E2 18800.653} C_VEL
LIN {X 0,Y 224.631,Z 778.358,A -85,B 0,C 180,E1 18809.325,E2 18809.325} C_VEL
LIN {X 0,Y 217.471,Z 791.222,A -85,B 0,C 180,E1 18818.979,E2 18818.979} C_VEL
LIN {X 0,Y 214.592,Z 797.048,A -85,B 0,C 180,E1 18826.334,E2 18826.334} C_VEL
LIN {X 0,Y 212.982,Z 800.245,A -85,B 0,C 180,E1 18835.154,E2 18835.154} C_VEL
LIN {X 0,Y 214.289,Z 799.428,A -85,B 0,C 180,E1 18844.285,E2 18844.285} C_VEL
LIN {X 0,Y 218.419,Z 794.124,A -85,B 0,C 180,E1 18853.696,E2 18853.696} C_VEL
LIN {X 0,Y 226.38,Z 783.428,A -85,B 0,C 180,E1 18863.185,E2 18863.185} C_VEL
LIN {X 0,Y 237.713,Z 768.457,A -85,B 0,C 180,E1 18871.246,E2 18871.246} C_VEL
LIN {X 0,Y 252.643,Z 747.829,A -85,B 0,C 180,E1 18878.393,E2 18878.393} C_VEL
LIN {X 0,Y 269.239,Z 722.063,A -85,B 0,C 180,E1 18884.259,E2 18884.259} C_VEL
LIN {X 0,Y 285.909,Z 691.241,A -85,B 0,C 180,E1 18888.858,E2 18888.858} C_VEL
LIN {X 0,Y 289.099,Z 683.63,A -85,B 0,C 180,E1 18889.931,E2 18889.931} C_VEL
LIN {X 0,Y 289.211,Z 667.075,A -85,B 0,C 180,E1 18895.162,E2 18895.162} C_VEL
LIN {X 0,Y 288.289,Z 654.086,A -85,B 0,C 180,E1 18901.017,E2 18901.017} C_VEL
LIN {X 0,Y 287.731,Z 647.915,A -85,B 0,C 180,E1 18906.045,E2 18906.045} C_VEL
LIN {X 0,Y 287.785,Z 647.91,A -85,B 0,C 180,E1 18912.13,E2 18912.13} C_VEL
LIN {X 0,Y 289.574,Z 654.25,A -85,B 0,C 180,E1 18918.242,E2 18918.242} C_VEL
LIN {X 0,Y 292.395,Z 666.59,A -85,B 0,C 180,E1 18923.981,E2 18923.981} C_VEL
LIN {X 0,Y 294.459,Z 682.414,A -85,B 0,C 180,E1 18928.834,E2 18928.834} C_VEL
LIN {X 0,Y 294.364,Z 687.624,A -85,B 0,C 180,E1 18929.998,E2 18929.998} C_VEL
LIN {X 0,Y 277.292,Z 724.07,A -85,B 0,C 180,E1 18933.916,E2 18933.916} C_VEL
LIN {X 0,Y 259.853,Z 755.097,A -85,B 0,C 180,E1 18939.044,E2 18939.044} C_VEL
LIN {X 0,Y 243.967,Z 780.452,A -85,B 0,C 180,E1 18945.269,E2 18945.269} C_VEL
LIN {X 0,Y 230.27,Z 801.715,A -85,B 0,C 180,E1 18952.973,E2 18952.973} C_VEL
LIN {X 0,Y 219.783,Z 819.367,A -85,B 0,C 180,E1 18962.629,E2 18962.629} C_VEL
LIN {X 0,Y 214.828,Z 830.684,A -85,B 0,C 180,E1 18972.324,E2 18972.324} C_VEL
LIN {X 0,Y 213.48,Z 836.985,A -85,B 0,C 180,E1 18981.876,E2 18981.876} C_VEL
LIN {X 0,Y 213.95,Z 838.593,A -85,B 0,C 180,E1 18990.003,E2 18990.003} C_VEL
LIN {X 0,Y 213.483,Z 836.569,A -85,B 0,C 180,E1 18998.13,E2 18998.13} C_VEL
LIN {X 0,Y 214.89,Z 829.688,A -85,B 0,C 180,E1 19007.711,E2 19007.711} C_VEL
LIN {X 0,Y 220.22,Z 816.471,A -85,B 0,C 180,E1 19017.979,E2 19017.979} C_VEL
LIN {X 0,Y 229.983,Z 798.194,A -85,B 0,C 180,E1 19027.009,E2 19027.009} C_VEL
LIN {X 0,Y 243.857,Z 773.798,A -85,B 0,C 180,E1 19034.982,E2 19034.982} C_VEL
LIN {X 0,Y 259.63,Z 744.193,A -85,B 0,C 180,E1 19041.357,E2 19041.357} C_VEL
LIN {X 0,Y 274.58,Z 712.083,A -85,B 0,C 180,E1 19045.948,E2 19045.948} C_VEL
LIN {X 0,Y 285.679,Z 682.969,A -85,B 0,C 180,E1 19048.883,E2 19048.883} C_VEL
LIN {X 0,Y 279.394,Z 659.06,A -85,B 0,C 180,E1 19054.378,E2 19054.378} C_VEL
LIN {X 0,Y 269.986,Z 634.792,A -85,B 0,C 180,E1 19061.159,E2 19061.159} C_VEL
LIN {X 0,Y 260.996,Z 616.808,A -85,B 0,C 180,E1 19067.779,E2 19067.779} C_VEL
LIN {X 0,Y 252.335,Z 601.003,A -85,B 0,C 180,E1 19075.471,E2 19075.471} C_VEL
LIN {X 0,Y 247.715,Z 593.848,A -85,B 0,C 180,E1 19080.713,E2 19080.713} C_VEL
LIN {X 0,Y 244.388,Z 588.135,A -85,B 0,C 180,E1 19086.305,E2 19086.305} C_VEL
LIN {X 0,Y 241.385,Z 587.12,A -85,B 0,C 180,E1 19098.179,E2 19098.179} C_VEL
LIN {X 0,Y 242.032,Z 587.766,A -85,B 0,C 180,E1 19102.164,E2 19102.164} C_VEL
LIN {X 0,Y 242.393,Z 591.828,A -85,B 0,C 180,E1 19105.101,E2 19105.101} C_VEL
LIN {X 0,Y 242.946,Z 600.872,A -85,B 0,C 180,E1 19109.322,E2 19109.322} C_VEL
LIN {X 0,Y 243.214,Z 601.295,A -85,B 0,C 180,E1 19109.832,E2 19109.832} C_VEL
LIN {X 0,Y 245.244,Z 604.375,A -85,B 0,C 180,E1 19113.035,E2 19113.035} C_VEL
LIN {X 0,Y 249.154,Z 611.981,A -85,B 0,C 180,E1 19118.328,E2 19118.328} C_VEL
LIN {X 0,Y 254.485,Z 622.374,A -85,B 0,C 180,E1 19124.021,E2 19124.021} C_VEL
LIN {X 0,Y 261.949,Z 639.329,A -85,B 0,C 180,E1 19131.07,E2 19131.07} C_VEL
LIN {X 0,Y 268.222,Z 660.717,A -85,B 0,C 180,E1 19137.804,E2 19137.804} C_VEL
LIN {X 0,Y 271.262,Z 679.386,A -85,B 0,C 180,E1 19142.798,E2 19142.798} C_VEL
LIN {X 0,Y 256.723,Z 711.587,A -85,B 0,C 180,E1 19147.307,E2 19147.307} C_VEL
LIN {X 0,Y 241.607,Z 739.624,A -85,B 0,C 180,E1 19153.207,E2 19153.207} C_VEL
LIN {X 0,Y 227.845,Z 762.436,A -85,B 0,C 180,E1 19160.465,E2 19160.465} C_VEL
LIN {X 0,Y 217.076,Z 779.551,A -85,B 0,C 180,E1 19168.815,E2 19168.815} C_VEL
LIN {X 0,Y 209.931,Z 791.726,A -85,B 0,C 180,E1 19178.263,E2 19178.263} C_VEL
LIN {X 0,Y 206.181,Z 798.795,A -85,B 0,C 180,E1 19188.081,E2 19188.081} C_VEL
LIN {X 0,Y 205.163,Z 801.168,A -85,B 0,C 180,E1 19198.14,E2 19198.14} C_VEL
LIN {X 0,Y 207.349,Z 799.406,A -85,B 0,C 180,E1 19206.894,E2 19206.894} C_VEL
LIN {X 0,Y 212.829,Z 792.637,A -85,B 0,C 180,E1 19217.13,E2 19217.13} C_VEL
LIN {X 0,Y 221.971,Z 781.279,A -85,B 0,C 180,E1 19226.261,E2 19226.261} C_VEL
LIN {X 0,Y 235.733,Z 764.054,A -85,B 0,C 180,E1 19234.685,E2 19234.685} C_VEL
LIN {X 0,Y 252.211,Z 741.764,A -85,B 0,C 180,E1 19241.611,E2 19241.611} C_VEL
LIN {X 0,Y 269.655,Z 714.683,A -85,B 0,C 180,E1 19247.096,E2 19247.096} C_VEL
LIN {X 0,Y 284.027,Z 687.659,A -85,B 0,C 180,E1 19250.856,E2 19250.856} C_VEL
LIN {X 0,Y 284.782,Z 671.694,A -85,B 0,C 180,E1 19256.228,E2 19256.228} C_VEL
LIN {X 0,Y 284.596,Z 661.408,A -85,B 0,C 180,E1 19261.03,E2 19261.03} C_VEL
LIN {X 0,Y 284.465,Z 655.132,A -85,B 0,C 180,E1 19266.114,E2 19266.114} C_VEL
LIN {X 0,Y 284.558,Z 655.256,A -85,B 0,C 180,E1 19272.27,E2 19272.27} C_VEL
LIN {X 0,Y 286.244,Z 661.916,A -85,B 0,C 180,E1 19278.399,E2 19278.399} C_VEL
LIN {X 0,Y 288.396,Z 673.966,A -85,B 0,C 180,E1 19283.945,E2 19283.945} C_VEL
LIN {X 0,Y 289.613,Z 689.429,A -85,B 0,C 180,E1 19288.665,E2 19288.665} C_VEL
LIN {X 0,Y 272.167,Z 725.355,A -85,B 0,C 180,E1 19292.692,E2 19292.692} C_VEL
LIN {X 0,Y 254.816,Z 754.865,A -85,B 0,C 180,E1 19297.625,E2 19297.625} C_VEL
LIN {X 0,Y 237.85,Z 780.61,A -85,B 0,C 180,E1 19304.052,E2 19304.052} C_VEL
LIN {X 0,Y 222.669,Z 802.76,A -85,B 0,C 180,E1 19312.42,E2 19312.42} C_VEL
LIN {X 0,Y 211.748,Z 820.173,A -85,B 0,C 180,E1 19322.617,E2 19322.617} C_VEL
LIN {X 0,Y 206.702,Z 831.167,A -85,B 0,C 180,E1 19333.024,E2 19333.024} C_VEL
LIN {X 0,Y 205.583,Z 836.297,A -85,B 0,C 180,E1 19341.561,E2 19341.561} C_VEL
LIN {X 0,Y 206.093,Z 837.874,A -85,B 0,C 180,E1 19350.003,E2 19350.003} C_VEL
LIN {X 0,Y 205.592,Z 835.807,A -85,B 0,C 180,E1 19358.445,E2 19358.445} C_VEL
LIN {X 0,Y 207.288,Z 828.474,A -85,B 0,C 180,E1 19368.781,E2 19368.781} C_VEL
LIN {X 0,Y 212.576,Z 816.316,A -85,B 0,C 180,E1 19378.505,E2 19378.505} C_VEL
LIN {X 0,Y 222.492,Z 798.698,A -85,B 0,C 180,E1 19387.623,E2 19387.623} C_VEL
LIN {X 0,Y 235.302,Z 777.138,A -85,B 0,C 180,E1 19395.105,E2 19395.105} C_VEL
LIN {X 0,Y 250.724,Z 749.861,A -85,B 0,C 180,E1 19401.487,E2 19401.487} C_VEL
LIN {X 0,Y 266.62,Z 717.981,A -85,B 0,C 180,E1 19406.454,E2 19406.454} C_VEL
LIN {X 0,Y 279.491,Z 686.595,A -85,B 0,C 180,E1 19409.758,E2 19409.758} C_VEL
LIN {X 0,Y 274.685,Z 665.272,A -85,B 0,C 180,E1 19414.779,E2 19414.779} C_VEL
LIN {X 0,Y 265.965,Z 640.916,A -85,B 0,C 180,E1 19421.793,E2 19421.793} C_VEL
LIN {X 0,Y 257.865,Z 623.725,A -85,B 0,C 180,E1 19428.262,E2 19428.262} C_VEL
LIN {X 0,Y 249.905,Z 608.249,A -85,B 0,C 180,E1 19435.969,E2 19435.969} C_VEL
LIN {X 0,Y 245.576,Z 601.043,A -85,B 0,C 180,E1 19441.401,E2 19441.401} C_VEL
LIN {X 0,Y 242.885,Z 595.891,A -85,B 0,C 180,E1 19446.224,E2 19446.224} C_VEL
LIN {X 0,Y 239.821,Z 594.862,A -85,B 0,C 180,E1 19458.301,E2 19458.301} C_VEL
LIN {X 0,Y 241.465,Z 596.844,A -85,B 0,C 180,E1 19465.301,E2 19465.301} C_VEL
LIN {X 0,Y 243.214,Z 601.295,A -85,B 0,C 180,E1 19469.832,E2 19469.832} C_VEL
LIN {X 0,Y 243.73,Z 605.287,A -85,B 0,C 180,E1 19471.658,E2 19471.658} C_VEL
LIN {X 0,Y 243.886,Z 614.221,A -85,B 0,C 180,E1 19474.503,E2 19474.503} C_VEL
LIN {X 0,Y 248.194,Z 622.741,A -85,B 0,C 180,E1 19480.191,E2 19480.191} C_VEL
LIN {X 0,Y 254.831,Z 638.033,A -85,B 0,C 180,E1 19487.558,E2 19487.558} C_VEL
LIN {X 0,Y 260.231,Z 654.119,A -85,B 0,C 180,E1 19493.515,E2 19493.515} C_VEL
LIN {X 0,Y 264.654,Z 675.637,A -85,B 0,C 180,E1 19499.986,E2 19499.986} C_VEL
LIN {X 0,Y 265.024,Z 683.098,A -85,B 0,C 180,E1 19501.881,E2 19501.881} C_VEL
LIN {X 0,Y 250.604,Z 713.519,A -85,B 0,C 180,E1 19506.251,E2 19506.251} C_VEL
LIN {X 0,Y 234.999,Z 741.261,A -85,B 0,C 180,E1 19512.238,E2 19512.238} C_VEL
LIN {X 0,Y 220.731,Z 763.786,A -85,B 0,C 180,E1 19519.659,E2 19519.659} C_VEL
LIN {X 0,Y 208.764,Z 781.86,A -85,B 0,C 180,E1 19529.004,E2 19529.004} C_VEL
LIN {X 0,Y 201.848,Z 793.23,A -85,B 0,C 180,E1 19538.596,E2 19538.596} C_VEL
LIN {X 0,Y 198.39,Z 799.419,A -85,B 0,C 180,E1 19547.71,E2 19547.71} C_VEL
LIN {X 0,Y 197.248,Z 801.911,A -85,B 0,C 180,E1 19557.32,E2 19557.32} C_VEL
LIN {X 0,Y 200.044,Z 799.71,A -85,B 0,C 180,E1 19568.482,E2 19568.482} C_VEL
LIN {X 0,Y 206.199,Z 792.644,A -85,B 0,C 180,E1 19578.862,E2 19578.862} C_VEL
LIN {X 0,Y 216.696,Z 780.544,A -85,B 0,C 180,E1 19588.41,E2 19588.41} C_VEL
LIN {X 0,Y 232.155,Z 762.242,A -85,B 0,C 180,E1 19597.085,E2 19597.085} C_VEL
LIN {X 0,Y 249.965,Z 739.053,A -85,B 0,C 180,E1 19603.941,E2 19603.941} C_VEL
LIN {X 0,Y 268.372,Z 710.852,A -85,B 0,C 180,E1 19609.276,E2 19609.276} C_VEL
LIN {X 0,Y 279.18,Z 690.858,A -85,B 0,C 180,E1 19612.087,E2 19612.087} C_VEL
LIN {X 0,Y 280.523,Z 675.447,A -85,B 0,C 180,E1 19617.714,E2 19617.714} C_VEL
LIN {X 0,Y 280.82,Z 665.54,A -85,B 0,C 180,E1 19623.105,E2 19623.105} C_VEL
LIN {X 0,Y 280.991,Z 662.237,A -85,B 0,C 180,E1 19626.19,E2 19626.19} C_VEL
LIN {X 0,Y 281.194,Z 662.548,A -85,B 0,C 180,E1 19632.419,E2 19632.419} C_VEL
LIN {X 0,Y 282.384,Z 668.405,A -85,B 0,C 180,E1 19637.919,E2 19637.919} C_VEL
LIN {X 0,Y 283.964,Z 679.728,A -85,B 0,C 180,E1 19643.335,E2 19643.335} C_VEL
LIN {X 0,Y 284.495,Z 692.955,A -85,B 0,C 180,E1 19647.588,E2 19647.588} C_VEL
LIN {X 0,Y 267.196,Z 726.65,A -85,B 0,C 180,E1 19651.425,E2 19651.425} C_VEL
LIN {X 0,Y 248.774,Z 756.43,A -85,B 0,C 180,E1 19656.518,E2 19656.518} C_VEL
LIN {X 0,Y 231.045,Z 781.874,A -85,B 0,C 180,E1 19663.109,E2 19663.109} C_VEL
LIN {X 0,Y 214.761,Z 804.3,A -85,B 0,C 180,E1 19672.065,E2 19672.065} C_VEL
LIN {X 0,Y 203.527,Z 821.255,A -85,B 0,C 180,E1 19682.889,E2 19682.889} C_VEL
LIN {X 0,Y 198.448,Z 832.096,A -85,B 0,C 180,E1 19694.569,E2 19694.569} C_VEL
LIN {X 0,Y 197.552,Z 836.263,A -85,B 0,C 180,E1 19703.42,E2 19703.42} C_VEL
LIN {X 0,Y 198.227,Z 837.155,A -85,B 0,C 180,E1 19710.003,E2 19710.003} C_VEL
LIN {X 0,Y 197.713,Z 835.04,A -85,B 0,C 180,E1 19718.784,E2 19718.784} C_VEL
LIN {X 0,Y 199.025,Z 829.341,A -85,B 0,C 180,E1 19727.658,E2 19727.658} C_VEL
LIN {X 0,Y 204.754,Z 816.548,A -85,B 0,C 180,E1 19738.813,E2 19738.813} C_VEL
LIN {X 0,Y 215.274,Z 798.729,A -85,B 0,C 180,E1 19748.474,E2 19748.474} C_VEL
LIN {X 0,Y 229.181,Z 776.407,A -85,B 0,C 180,E1 19756.413,E2 19756.413} C_VEL
LIN {X 0,Y 244.788,Z 749.855,A -85,B 0,C 180,E1 19762.712,E2 19762.712} C_VEL
LIN {X 0,Y 260.503,Z 719.506,A -85,B 0,C 180,E1 19767.523,E2 19767.523} C_VEL
LIN {X 0,Y 273.666,Z 688.639,A -85,B 0,C 180,E1 19770.882,E2 19770.882} C_VEL
LIN {X 0,Y 268.161,Z 665.637,A -85,B 0,C 180,E1 19776.779,E2 19776.779} C_VEL
LIN {X 0,Y 260.97,Z 644.894,A -85,B 0,C 180,E1 19783.17,E2 19783.17} C_VEL
LIN {X 0,Y 253.077,Z 626.97,A -85,B 0,C 180,E1 19790.319,E2 19790.319} C_VEL
LIN {X 0,Y 246.414,Z 614.093,A -85,B 0,C 180,E1 19797.553,E2 19797.553} C_VEL
LIN {X 0,Y 243.263,Z 608.274,A -85,B 0,C 180,E1 19801.991,E2 19801.991} C_VEL
LIN {X 0,Y 240.636,Z 603.441,A -85,B 0,C 180,E1 19807.173,E2 19807.173} C_VEL
LIN {X 0,Y 238.148,Z 602.752,A -85,B 0,C 180,E1 19819.483,E2 19819.483} C_VEL
LIN {X 0,Y 239.452,Z 604.534,A -85,B 0,C 180,E1 19825.099,E2 19825.099} C_VEL
LIN {X 0,Y 242.918,Z 612.063,A -85,B 0,C 180,E1 19832.882,E2 19832.882} C_VEL
LIN {X 0,Y 243.886,Z 614.221,A -85,B 0,C 180,E1 19834.503,E2 19834.503} C_VEL
LIN {X 0,Y 244.154,Z 621.267,A -85,B 0,C 180,E1 19836.737,E2 19836.737} C_VEL
LIN {X 0,Y 244.472,Z 628.299,A -85,B 0,C 180,E1 19838.973,E2 19838.973} C_VEL
LIN {X 0,Y 250.545,Z 643.617,A -85,B 0,C 180,E1 19846.718,E2 19846.718} C_VEL
LIN {X 0,Y 255.769,Z 661.046,A -85,B 0,C 180,E1 19853.321,E2 19853.321} C_VEL
LIN {X 0,Y 259.164,Z 681.213,A -85,B 0,C 180,E1 19859.577,E2 19859.577} C_VEL
LIN {X 0,Y 259.136,Z 685.862,A -85,B 0,C 180,E1 19860.785,E2 19860.785} C_VEL
LIN {X 0,Y 243.997,Z 716.467,A -85,B 0,C 180,E1 19865.323,E2 19865.323} C_VEL
LIN {X 0,Y 227.487,Z 744.349,A -85,B 0,C 180,E1 19871.631,E2 19871.631} C_VEL
LIN {X 0,Y 212.82,Z 766.235,A -85,B 0,C 180,E1 19879.27,E2 19879.27} C_VEL
LIN {X 0,Y 201.803,Z 782.167,A -85,B 0,C 180,E1 19887.854,E2 19887.854} C_VEL
LIN {X 0,Y 194.336,Z 793.719,A -85,B 0,C 180,E1 19897.807,E2 19897.807} C_VEL
LIN {X 0,Y 190.346,Z 800.372,A -85,B 0,C 180,E1 19908.114,E2 19908.114} C_VEL
LIN {X 0,Y 189.44,Z 802.605,A -85,B 0,C 180,E1 19918.913,E2 19918.913} C_VEL
LIN {X 0,Y 192.324,Z 800.58,A -85,B 0,C 180,E1 19928.876,E2 19928.876} C_VEL
LIN {X 0,Y 198.655,Z 793.888,A -85,B 0,C 180,E1 19939.425,E2 19939.425} C_VEL
LIN {X 0,Y 210.662,Z 781,A -85,B 0,C 180,E1 19949.953,E2 19949.953} C_VEL
LIN {X 0,Y 226.865,Z 762.921,A -85,B 0,C 180,E1 19958.618,E2 19958.618} C_VEL
LIN {X 0,Y 245.993,Z 739.136,A -85,B 0,C 180,E1 19965.632,E2 19965.632} C_VEL
LIN {X 0,Y 264.86,Z 711.299,A -85,B 0,C 180,E1 19970.839,E2 19970.839} C_VEL
LIN {X 0,Y 273.719,Z 696.212,A -85,B 0,C 180,E1 19972.885,E2 19972.885} C_VEL
LIN {X 0,Y 275.655,Z 685.805,A -85,B 0,C 180,E1 19976.418,E2 19976.418} C_VEL
LIN {X 0,Y 276.729,Z 674.963,A -85,B 0,C 180,E1 19981.588,E2 19981.588} C_VEL
LIN {X 0,Y 277.376,Z 669.308,A -85,B 0,C 180,E1 19986.271,E2 19986.271} C_VEL
LIN {X 0,Y 277.627,Z 669.758,A -85,B 0,C 180,E1 19992.581,E2 19992.581} C_VEL
LIN {X 0,Y 278.616,Z 675.993,A -85,B 0,C 180,E1 19998.168,E2 19998.168} C_VEL
LIN {X 0,Y 279.618,Z 688.577,A -85,B 0,C 180,E1 20003.896,E2 20003.896} C_VEL
LIN {X 0,Y 279.31,Z 697.19,A -85,B 0,C 180,E1 20006.576,E2 20006.576} C_VEL
LIN {X 0,Y 259.895,Z 732.084,A -85,B 0,C 180,E1 20010.682,E2 20010.682} C_VEL
LIN {X 0,Y 240.467,Z 761.311,A -85,B 0,C 180,E1 20016.082,E2 20016.082} C_VEL
LIN {X 0,Y 221.559,Z 786.673,A -85,B 0,C 180,E1 20023.337,E2 20023.337} C_VEL
LIN {X 0,Y 205.479,Z 807.518,A -85,B 0,C 180,E1 20032.713,E2 20032.713} C_VEL
LIN {X 0,Y 195.021,Z 822.657,A -85,B 0,C 180,E1 20043.586,E2 20043.586} C_VEL
LIN {X 0,Y 190.671,Z 831.437,A -85,B 0,C 180,E1 20053.922,E2 20053.922} C_VEL
LIN {X 0,Y 189.819,Z 834.912,A -85,B 0,C 180,E1 20060.855,E2 20060.855} C_VEL
LIN {X 0,Y 190.362,Z 836.434,A -85,B 0,C 180,E1 20070.003,E2 20070.003} C_VEL
LIN {X 0,Y 189.833,Z 834.27,A -85,B 0,C 180,E1 20079.151,E2 20079.151} C_VEL
LIN {X 0,Y 191.443,Z 828.071,A -85,B 0,C 180,E1 20088.86,E2 20088.86} C_VEL
LIN {X 0,Y 197.46,Z 815.818,A -85,B 0,C 180,E1 20099.788,E2 20099.788} C_VEL
LIN {X 0,Y 208.856,Z 797.603,A -85,B 0,C 180,E1 20109.888,E2 20109.888} C_VEL
LIN {X 0,Y 223.538,Z 775.09,A -85,B 0,C 180,E1 20117.955,E2 20117.955} C_VEL
LIN {X 0,Y 239.998,Z 748.012,A -85,B 0,C 180,E1 20124.341,E2 20124.341} C_VEL
LIN {X 0,Y 256.817,Z 716.309,A -85,B 0,C 180,E1 20129.247,E2 20129.247} C_VEL
LIN {X 0,Y 267.692,Z 691.296,A -85,B 0,C 180,E1 20131.997,E2 20131.997} C_VEL
LIN {X 0,Y 263.001,Z 670.263,A -85,B 0,C 180,E1 20137.635,E2 20137.635} C_VEL
LIN {X 0,Y 255.994,Z 648.722,A -85,B 0,C 180,E1 20144.592,E2 20144.592} C_VEL
LIN {X 0,Y 249.345,Z 633.019,A -85,B 0,C 180,E1 20151.271,E2 20151.271} C_VEL
LIN {X 0,Y 243.587,Z 621.01,A -85,B 0,C 180,E1 20158.218,E2 20158.218} C_VEL
LIN {X 0,Y 240.846,Z 615.493,A -85,B 0,C 180,E1 20162.586,E2 20162.586} C_VEL
LIN {X 0,Y 238.689,Z 611.068,A -85,B 0,C 180,E1 20167.232,E2 20167.232} C_VEL
LIN {X 0,Y 236.246,Z 610.408,A -85,B 0,C 180,E1 20179.556,E2 20179.556} C_VEL
LIN {X 0,Y 237.282,Z 612.065,A -85,B 0,C 180,E1 20184.767,E2 20184.767} C_VEL
LIN {X 0,Y 240.367,Z 619.433,A -85,B 0,C 180,E1 20192.554,E2 20192.554} C_VEL
LIN {X 0,Y 244.472,Z 628.299,A -85,B 0,C 180,E1 20198.973,E2 20198.973} C_VEL
LIN {X 0,Y 245.593,Z 634.949,A -85,B 0,C 180,E1 20201.586,E2 20201.586} C_VEL
LIN {X 0,Y 246.081,Z 648.791,A -85,B 0,C 180,E1 20205.657,E2 20205.657} C_VEL
LIN {X 0,Y 250.655,Z 665.821,A -85,B 0,C 180,E1 20212.457,E2 20212.457} C_VEL
LIN {X 0,Y 253.444,Z 685.302,A -85,B 0,C 180,E1 20218.763,E2 20218.763} C_VEL
LIN {X 0,Y 252.711,Z 690.073,A -85,B 0,C 180,E1 20219.821,E2 20219.821} C_VEL
LIN {X 0,Y 236.833,Z 720.304,A -85,B 0,C 180,E1 20224.524,E2 20224.524} C_VEL
LIN {X 0,Y 219.938,Z 747.336,A -85,B 0,C 180,E1 20230.977,E2 20230.977} C_VEL
LIN {X 0,Y 204.142,Z 769.76,A -85,B 0,C 180,E1 20239.347,E2 20239.347} C_VEL
LIN {X 0,Y 192.678,Z 785.628,A -85,B 0,C 180,E1 20248.875,E2 20248.875} C_VEL
LIN {X 0,Y 185.648,Z 796.177,A -85,B 0,C 180,E1 20259.352,E2 20259.352} C_VEL
LIN {X 0,Y 182.121,Z 801.64,A -85,B 0,C 180,E1 20269.352,E2 20269.352} C_VEL
LIN {X 0,Y 181.679,Z 803.313,A -85,B 0,C 180,E1 20279.887,E2 20279.887} C_VEL
LIN {X 0,Y 185.191,Z 800.852,A -85,B 0,C 180,E1 20290.678,E2 20290.678} C_VEL
LIN {X 0,Y 192.525,Z 793.706,A -85,B 0,C 180,E1 20301.604,E2 20301.604} C_VEL
LIN {X 0,Y 205.944,Z 780.339,A -85,B 0,C 180,E1 20312.306,E2 20312.306} C_VEL
LIN {X 0,Y 223.514,Z 761.759,A -85,B 0,C 180,E1 20320.932,E2 20320.932} C_VEL
LIN {X 0,Y 243.77,Z 737.222,A -85,B 0,C 180,E1 20327.838,E2 20327.838} C_VEL
LIN {X 0,Y 262.731,Z 709.948,A -85,B 0,C 180,E1 20332.721,E2 20332.721} C_VEL
LIN {X 0,Y 269.067,Z 699.538,A -85,B 0,C 180,E1 20334.103,E2 20334.103} C_VEL
LIN {X 0,Y 271.666,Z 687.332,A -85,B 0,C 180,E1 20338.844,E2 20338.844} C_VEL
LIN {X 0,Y 273.078,Z 678.377,A -85,B 0,C 180,E1 20344.218,E2 20344.218} C_VEL
LIN {X 0,Y 273.464,Z 676.123,A -85,B 0,C 180,E1 20346.674,E2 20346.674} C_VEL
LIN {X 0,Y 273.797,Z 676.881,A -85,B 0,C 180,E1 20352.76,E2 20352.76} C_VEL
LIN {X 0,Y 274.526,Z 683.242,A -85,B 0,C 180,E1 20358.222,E2 20358.222} C_VEL
LIN {X 0,Y 274.868,Z 694.001,A -85,B 0,C 180,E1 20363.241,E2 20363.241} C_VEL
LIN {X 0,Y 274.181,Z 700.872,A -85,B 0,C 180,E1 20365.413,E2 20365.413} C_VEL
LIN {X 0,Y 255.204,Z 733.214,A -85,B 0,C 180,E1 20369.294,E2 20369.294} C_VEL
LIN {X 0,Y 235.162,Z 761.952,A -85,B 0,C 180,E1 20374.675,E2 20374.675} C_VEL
LIN {X 0,Y 215.558,Z 786.867,A -85,B 0,C 180,E1 20381.956,E2 20381.956} C_VEL
LIN {X 0,Y 199.012,Z 807.028,A -85,B 0,C 180,E1 20391.281,E2 20391.281} C_VEL
LIN {X 0,Y 187.371,Z 822.656,A -85,B 0,C 180,E1 20403.022,E2 20403.022} C_VEL
LIN {X 0,Y 182.415,Z 832.184,A -85,B 0,C 180,E1 20415.634,E2 20415.634} C_VEL
LIN {X 0,Y 181.891,Z 835.383,A -85,B 0,C 180,E1 20425.245,E2 20425.245} C_VEL
LIN {X 0,Y 182.493,Z 835.712,A -85,B 0,C 180,E1 20430.004,E2 20430.004} C_VEL
LIN {X 0,Y 181.99,Z 833.496,A -85,B 0,C 180,E1 20439.549,E2 20439.549} C_VEL
LIN {X 0,Y 184.026,Z 826.579,A -85,B 0,C 180,E1 20450.399,E2 20450.399} C_VEL
LIN {X 0,Y 190.383,Z 814.826,A -85,B 0,C 180,E1 20461.015,E2 20461.015} C_VEL
LIN {X 0,Y 202.593,Z 796.454,A -85,B 0,C 180,E1 20471.385,E2 20471.385} C_VEL
LIN {X 0,Y 218.041,Z 773.73,A -85,B 0,C 180,E1 20479.582,E2 20479.582} C_VEL
LIN {X 0,Y 236.023,Z 745.16,A -85,B 0,C 180,E1 20486.223,E2 20486.223} C_VEL
LIN {X 0,Y 254.029,Z 711.51,A -85,B 0,C 180,E1 20491.192,E2 20491.192} C_VEL
LIN {X 0,Y 261.701,Z 693.903,A -85,B 0,C 180,E1 20493.138,E2 20493.138} C_VEL
LIN {X 0,Y 257.099,Z 672.06,A -85,B 0,C 180,E1 20499.356,E2 20499.356} C_VEL
LIN {X 0,Y 250.718,Z 651.638,A -85,B 0,C 180,E1 20506.477,E2 20506.477} C_VEL
LIN {X 0,Y 244.179,Z 635.294,A -85,B 0,C 180,E1 20514.066,E2 20514.066} C_VEL
LIN {X 0,Y 238.641,Z 623.262,A -85,B 0,C 180,E1 20522.429,E2 20522.429} C_VEL
LIN {X 0,Y 236.485,Z 618.652,A -85,B 0,C 180,E1 20527.3,E2 20527.3} C_VEL
LIN {X 0,Y 234.038,Z 617.999,A -85,B 0,C 180,E1 20539.748,E2 20539.748} C_VEL
LIN {X 0,Y 234.927,Z 619.664,A -85,B 0,C 180,E1 20544.563,E2 20544.563} C_VEL
LIN {X 0,Y 237.529,Z 626.666,A -85,B 0,C 180,E1 20552.21,E2 20552.21} C_VEL
LIN {X 0,Y 241.583,Z 636.567,A -85,B 0,C 180,E1 20559.288,E2 20559.288} C_VEL
LIN {X 0,Y 246.081,Z 648.791,A -85,B 0,C 180,E1 20565.657,E2 20565.657} C_VEL
LIN {X 0,Y 246.54,Z 656.754,A -85,B 0,C 180,E1 20568.085,E2 20568.085} C_VEL
LIN {X 0,Y 245.772,Z 671.625,A -85,B 0,C 180,E1 20571.928,E2 20571.928} C_VEL
LIN {X 0,Y 247.808,Z 691.007,A -85,B 0,C 180,E1 20578.41,E2 20578.41} C_VEL
LIN {X 0,Y 230.923,Z 722.049,A -85,B 0,C 180,E1 20583.301,E2 20583.301} C_VEL
LIN {X 0,Y 214.509,Z 747.372,A -85,B 0,C 180,E1 20589.403,E2 20589.403} C_VEL
LIN {X 0,Y 198.772,Z 768.849,A -85,B 0,C 180,E1 20597.39,E2 20597.39} C_VEL
LIN {X 0,Y 185.673,Z 786.004,A -85,B 0,C 180,E1 20607.668,E2 20607.668} C_VEL
LIN {X 0,Y 178.708,Z 795.688,A -85,B 0,C 180,E1 20617.273,E2 20617.273} C_VEL
LIN {X 0,Y 174.506,Z 801.933,A -85,B 0,C 180,E1 20628.146,E2 20628.146} C_VEL
LIN {X 0,Y 174.017,Z 804.018,A -85,B 0,C 180,E1 20641.348,E2 20641.348} C_VEL
LIN {X 0,Y 178.211,Z 801.141,A -85,B 0,C 180,E1 20652.636,E2 20652.636} C_VEL
LIN {X 0,Y 187.853,Z 792.548,A -85,B 0,C 180,E1 20665.002,E2 20665.002} C_VEL
LIN {X 0,Y 203.187,Z 778.089,A -85,B 0,C 180,E1 20675.642,E2 20675.642} C_VEL
LIN {X 0,Y 221.979,Z 758.906,A -85,B 0,C 180,E1 20683.835,E2 20683.835} C_VEL
LIN {X 0,Y 242.804,Z 734.306,A -85,B 0,C 180,E1 20690.295,E2 20690.295} C_VEL
LIN {X 0,Y 263.456,Z 704.725,A -85,B 0,C 180,E1 20695.137,E2 20695.137} C_VEL
LIN {X 0,Y 264.737,Z 702.542,A -85,B 0,C 180,E1 20695.445,E2 20695.445} C_VEL
LIN {X 0,Y 267.659,Z 690.434,A -85,B 0,C 180,E1 20700.834,E2 20700.834} C_VEL
LIN {X 0,Y 269.106,Z 684.07,A -85,B 0,C 180,E1 20705.321,E2 20705.321} C_VEL
LIN {X 0,Y 269.51,Z 682.752,A -85,B 0,C 180,E1 20709.695,E2 20709.695} C_VEL
LIN {X 0,Y 269.983,Z 685.828,A -85,B 0,C 180,E1 20715.056,E2 20715.056} C_VEL
LIN {X 0,Y 270.194,Z 694.575,A -85,B 0,C 180,E1 20720.48,E2 20720.48} C_VEL
LIN {X 0,Y 269.315,Z 704.317,A -85,B 0,C 180,E1 20724.193,E2 20724.193} C_VEL
LIN {X 0,Y 248.567,Z 737.586,A -85,B 0,C 180,E1 20728.33,E2 20728.33} C_VEL
LIN {X 0,Y 225.94,Z 767.727,A -85,B 0,C 180,E1 20734.435,E2 20734.435} C_VEL
LIN {X 0,Y 205.044,Z 792.42,A -85,B 0,C 180,E1 20742.618,E2 20742.618} C_VEL
LIN {X 0,Y 189.211,Z 810.546,A -85,B 0,C 180,E1 20752.3,E2 20752.3} C_VEL
LIN {X 0,Y 178.137,Z 824.847,A -85,B 0,C 180,E1 20764.945,E2 20764.945} C_VEL
LIN {X 0,Y 174.292,Z 832.593,A -85,B 0,C 180,E1 20777.503,E2 20777.503} C_VEL
LIN {X 0,Y 174.004,Z 834.676,A -85,B 0,C 180,E1 20785.029,E2 20785.029} C_VEL
LIN {X 0,Y 174.599,Z 834.987,A -85,B 0,C 180,E1 20790.004,E2 20790.004} C_VEL
LIN {X 0,Y 174.118,Z 832.716,A -85,B 0,C 180,E1 20799.985,E2 20799.985} C_VEL
LIN {X 0,Y 176.436,Z 825.699,A -85,B 0,C 180,E1 20811.319,E2 20811.319} C_VEL
LIN {X 0,Y 183.377,Z 813.81,A -85,B 0,C 180,E1 20822.34,E2 20822.34} C_VEL
LIN {X 0,Y 196.459,Z 795.28,A -85,B 0,C 180,E1 20832.981,E2 20832.981} C_VEL
LIN {X 0,Y 212.767,Z 772.356,A -85,B 0,C 180,E1 20841.28,E2 20841.28} C_VEL
LIN {X 0,Y 231.542,Z 743.498,A -85,B 0,C 180,E1 20847.918,E2 20847.918} C_VEL
LIN {X 0,Y 249.388,Z 710.977,A -85,B 0,C 180,E1 20852.664,E2 20852.664} C_VEL
LIN {X 0,Y 255.772,Z 696.397,A -85,B 0,C 180,E1 20854.351,E2 20854.351} C_VEL
LIN {X 0,Y 251.6,Z 675.201,A -85,B 0,C 180,E1 20860.74,E2 20860.74} C_VEL
LIN {X 0,Y 245.873,Z 655.619,A -85,B 0,C 180,E1 20867.99,E2 20867.99} C_VEL
LIN {X 0,Y 239.581,Z 639.359,A -85,B 0,C 180,E1 20876.36,E2 20876.36} C_VEL
LIN {X 0,Y 236.516,Z 631.349,A -85,B 0,C 180,E1 20881.797,E2 20881.797} C_VEL
LIN {X 0,Y 234.15,Z 626.177,A -85,B 0,C 180,E1 20887.373,E2 20887.373} C_VEL
LIN {X 0,Y 231.613,Z 625.449,A -85,B 0,C 180,E1 20898.974,E2 20898.974} C_VEL
LIN {X 0,Y 232.22,Z 626.019,A -85,B 0,C 180,E1 20902.908,E2 20902.908} C_VEL
LIN {X 0,Y 234.593,Z 633.887,A -85,B 0,C 180,E1 20911.874,E2 20911.874} C_VEL
LIN {X 0,Y 238.29,Z 644.093,A -85,B 0,C 180,E1 20919.242,E2 20919.242} C_VEL
LIN {X 0,Y 242.634,Z 657.884,A -85,B 0,C 180,E1 20926.38,E2 20926.38} C_VEL
LIN {X 0,Y 245.772,Z 671.625,A -85,B 0,C 180,E1 20931.928,E2 20931.928} C_VEL
LIN {X 0,Y 244.042,Z 680.259,A -85,B 0,C 180,E1 20933.753,E2 20933.753} C_VEL
LIN {X 0,Y 241.823,Z 689.061,A -85,B 0,C 180,E1 20935.584,E2 20935.584} C_VEL
LIN {X 0,Y 241.588,Z 694.798,A -85,B 0,C 180,E1 20937.341,E2 20937.341} C_VEL
LIN {X 0,Y 225.116,Z 723.748,A -85,B 0,C 180,E1 20942.012,E2 20942.012} C_VEL
LIN {X 0,Y 207.063,Z 750.314,A -85,B 0,C 180,E1 20948.627,E2 20948.627} C_VEL
LIN {X 0,Y 190.063,Z 772.267,A -85,B 0,C 180,E1 20957.385,E2 20957.385} C_VEL
LIN {X 0,Y 177.624,Z 787.763,A -85,B 0,C 180,E1 20967.562,E2 20967.562} C_VEL
LIN {X 0,Y 170.585,Z 797.169,A -85,B 0,C 180,E1 20977.621,E2 20977.621} C_VEL
LIN {X 0,Y 167.299,Z 801.787,A -85,B 0,C 180,E1 20985.696,E2 20985.696} C_VEL
LIN {X 0,Y 165.657,Z 804.667,A -85,B 0,C 180,E1 20997.09,E2 20997.09} C_VEL
LIN {X 0,Y 168.422,Z 803.557,A -85,B 0,C 180,E1 21008.838,E2 21008.838} C_VEL
LIN {X 0,Y 175.547,Z 798.01,A -85,B 0,C 180,E1 21020.676,E2 21020.676} C_VEL
LIN {X 0,Y 188.259,Z 787.245,A -85,B 0,C 180,E1 21031.843,E2 21031.843} C_VEL
LIN {X 0,Y 206.783,Z 770.408,A -85,B 0,C 180,E1 21041.555,E2 21041.555} C_VEL
LIN {X 0,Y 229.027,Z 747.216,A -85,B 0,C 180,E1 21049.247,E2 21049.247} C_VEL
LIN {X 0,Y 250.196,Z 720.776,A -85,B 0,C 180,E1 21054.606,E2 21054.606} C_VEL
LIN {X 0,Y 260.16,Z 706.316,A -85,B 0,C 180,E1 21056.703,E2 21056.703} C_VEL
LIN {X 0,Y 263.258,Z 695.89,A -85,B 0,C 180,E1 21061.669,E2 21061.669} C_VEL
LIN {X 0,Y 265.23,Z 689.817,A -85,B 0,C 180,E1 21066.56,E2 21066.56} C_VEL
LIN {X 0,Y 265.339,Z 689.524,A -85,B 0,C 180,E1 21069.849,E2 21069.849} C_VEL
LIN {X 0,Y 265.709,Z 692.728,A -85,B 0,C 180,E1 21075.111,E2 21075.111} C_VEL
LIN {X 0,Y 265.457,Z 700.429,A -85,B 0,C 180,E1 21079.966,E2 21079.966} C_VEL
LIN {X 0,Y 264.892,Z 706.951,A -85,B 0,C 180,E1 21082.749,E2 21082.749} C_VEL
LIN {X 0,Y 243.421,Z 739.718,A -85,B 0,C 180,E1 21086.99,E2 21086.99} C_VEL
LIN {X 0,Y 220.466,Z 768.718,A -85,B 0,C 180,E1 21092.999,E2 21092.999} C_VEL
LIN {X 0,Y 199.567,Z 792.082,A -85,B 0,C 180,E1 21100.88,E2 21100.88} C_VEL
LIN {X 0,Y 182.928,Z 809.874,A -85,B 0,C 180,E1 21110.586,E2 21110.586} C_VEL
LIN {X 0,Y 171.634,Z 823.128,A -85,B 0,C 180,E1 21122.433,E2 21122.433} C_VEL
LIN {X 0,Y 166.862,Z 830.863,A -85,B 0,C 180,E1 21134.262,E2 21134.262} C_VEL
LIN {X 0,Y 166.109,Z 833.972,A -85,B 0,C 180,E1 21144.792,E2 21144.792} C_VEL
LIN {X 0,Y 166.727,Z 834.263,A -85,B 0,C 180,E1 21150.004,E2 21150.004} C_VEL
LIN {X 0,Y 166.253,Z 831.93,A -85,B 0,C 180,E1 21160.463,E2 21160.463} C_VEL
LIN {X 0,Y 168.887,Z 824.8,A -85,B 0,C 180,E1 21172.322,E2 21172.322} C_VEL
LIN {X 0,Y 177.657,Z 811.15,A -85,B 0,C 180,E1 21184.988,E2 21184.988} C_VEL
LIN {X 0,Y 192.241,Z 791.752,A -85,B 0,C 180,E1 21195.753,E2 21195.753} C_VEL
LIN {X 0,Y 210.396,Z 767.147,A -85,B 0,C 180,E1 21204.107,E2 21204.107} C_VEL
LIN {X 0,Y 229.236,Z 738.459,A -85,B 0,C 180,E1 21210.245,E2 21210.245} C_VEL
LIN {X 0,Y 246.754,Z 706.54,A -85,B 0,C 180,E1 21214.628,E2 21214.628} C_VEL
LIN {X 0,Y 249.875,Z 699.149,A -85,B 0,C 180,E1 21215.552,E2 21215.552} C_VEL
LIN {X 0,Y 245.951,Z 677.249,A -85,B 0,C 180,E1 21222.57,E2 21222.57} C_VEL
LIN {X 0,Y 241.295,Z 660.587,A -85,B 0,C 180,E1 21229.159,E2 21229.159} C_VEL
LIN {X 0,Y 235.976,Z 645.576,A -85,B 0,C 180,E1 21237.221,E2 21237.221} C_VEL
LIN {X 0,Y 232.794,Z 637.293,A -85,B 0,C 180,E1 21243.685,E2 21243.685} C_VEL
LIN {X 0,Y 231.478,Z 633.722,A -85,B 0,C 180,E1 21247.458,E2 21247.458} C_VEL
LIN {X 0,Y 229.053,Z 632.94,A -85,B 0,C 180,E1 21259.195,E2 21259.195} C_VEL
LIN {X 0,Y 229.603,Z 633.821,A -85,B 0,C 180,E1 21263.185,E2 21263.185} C_VEL
LIN {X 0,Y 231.669,Z 641.706,A -85,B 0,C 180,E1 21272.132,E2 21272.132} C_VEL
LIN {X 0,Y 235.137,Z 652.634,A -85,B 0,C 180,E1 21279.872,E2 21279.872} C_VEL
LIN {X 0,Y 238.741,Z 666.164,A -85,B 0,C 180,E1 21286.832,E2 21286.832} C_VEL
LIN {X 0,Y 241.42,Z 682.76,A -85,B 0,C 180,E1 21293.404,E2 21293.404} C_VEL
LIN {X 0,Y 241.823,Z 689.061,A -85,B 0,C 180,E1 21295.584,E2 21295.584} C_VEL
LIN {X 0,Y 239.839,Z 694.442,A -85,B 0,C 180,E1 21296.538,E2 21296.538} C_VEL
LIN {X 0,Y 230.129,Z 707.989,A -85,B 0,C 180,E1 21297.567,E2 21297.567} C_VEL
LIN {X 0,Y 212.052,Z 736.54,A -85,B 0,C 180,E1 21303.125,E2 21303.125} C_VEL
LIN {X 0,Y 193.514,Z 761.019,A -85,B 0,C 180,E1 21310.642,E2 21310.642} C_VEL
LIN {X 0,Y 177.587,Z 780.069,A -85,B 0,C 180,E1 21320.212,E2 21320.212} C_VEL
LIN {X 0,Y 165.933,Z 794,A -85,B 0,C 180,E1 21332.048,E2 21332.048} C_VEL
LIN {X 0,Y 160.054,Z 801.642,A -85,B 0,C 180,E1 21343.629,E2 21343.629} C_VEL
LIN {X 0,Y 157.883,Z 804.659,A -85,B 0,C 180,E1 21352.473,E2 21352.473} C_VEL
LIN {X 0,Y 159.004,Z 805.25,A -85,B 0,C 180,E1 21364.705,E2 21364.705} C_VEL
LIN {X 0,Y 164.827,Z 801.624,A -85,B 0,C 180,E1 21377.083,E2 21377.083} C_VEL
LIN {X 0,Y 177.566,Z 791.877,A -85,B 0,C 180,E1 21390.24,E2 21390.24} C_VEL
LIN {X 0,Y 196.096,Z 776.537,A -85,B 0,C 180,E1 21400.865,E2 21400.865} C_VEL
LIN {X 0,Y 217.786,Z 756.007,A -85,B 0,C 180,E1 21408.868,E2 21408.868} C_VEL
LIN {X 0,Y 239.478,Z 731.67,A -85,B 0,C 180,E1 21414.607,E2 21414.607} C_VEL
LIN {X 0,Y 255.158,Z 710.82,A -85,B 0,C 180,E1 21417.867,E2 21417.867} C_VEL
LIN {X 0,Y 258.326,Z 702.655,A -85,B 0,C 180,E1 21421.701,E2 21421.701} C_VEL
LIN {X 0,Y 260.765,Z 696.404,A -85,B 0,C 180,E1 21426.672,E2 21426.672} C_VEL
LIN {X 0,Y 260.944,Z 696.422,A -85,B 0,C 180,E1 21430.565,E2 21430.565} C_VEL
LIN {X 0,Y 261.158,Z 699.734,A -85,B 0,C 180,E1 21435.381,E2 21435.381} C_VEL
LIN {X 0,Y 260.426,Z 708.112,A -85,B 0,C 180,E1 21440.369,E2 21440.369} C_VEL
LIN {X 0,Y 259.108,Z 712.292,A -85,B 0,C 180,E1 21441.728,E2 21441.728} C_VEL
LIN {X 0,Y 236.977,Z 743.761,A -85,B 0,C 180,E1 21445.921,E2 21445.921} C_VEL
LIN {X 0,Y 213.497,Z 771.655,A -85,B 0,C 180,E1 21451.993,E2 21451.993} C_VEL
LIN {X 0,Y 190.047,Z 796.1,A -85,B 0,C 180,E1 21461.039,E2 21461.039} C_VEL
LIN {X 0,Y 172.467,Z 813.729,A -85,B 0,C 180,E1 21472.236,E2 21472.236} C_VEL
LIN {X 0,Y 161.952,Z 825.599,A -85,B 0,C 180,E1 21485.214,E2 21485.214} C_VEL
LIN {X 0,Y 158.332,Z 832.155,A -85,B 0,C 180,E1 21499.016,E2 21499.016} C_VEL
LIN {X 0,Y 158.854,Z 833.538,A -85,B 0,C 180,E1 21510.004,E2 21510.004} C_VEL
LIN {X 0,Y 158.395,Z 831.138,A -85,B 0,C 180,E1 21520.988,E2 21520.988} C_VEL
LIN {X 0,Y 162.023,Z 822.855,A -85,B 0,C 180,E1 21534.783,E2 21534.783} C_VEL
LIN {X 0,Y 172.498,Z 808.031,A -85,B 0,C 180,E1 21548.014,E2 21548.014} C_VEL
LIN {X 0,Y 188.568,Z 787.938,A -85,B 0,C 180,E1 21558.616,E2 21558.616} C_VEL
LIN {X 0,Y 207.145,Z 763.491,A -85,B 0,C 180,E1 21566.54,E2 21566.54} C_VEL
LIN {X 0,Y 227.26,Z 733.42,A -85,B 0,C 180,E1 21572.587,E2 21572.587} C_VEL
LIN {X 0,Y 244.059,Z 701.982,A -85,B 0,C 180,E1 21576.78,E2 21576.78} C_VEL
LIN {X 0,Y 240.498,Z 680.569,A -85,B 0,C 180,E1 21584.04,E2 21584.04} C_VEL
LIN {X 0,Y 236.464,Z 664.698,A -85,B 0,C 180,E1 21590.791,E2 21590.791} C_VEL
LIN {X 0,Y 231.927,Z 650.359,A -85,B 0,C 180,E1 21599.037,E2 21599.037} C_VEL
LIN {X 0,Y 228.633,Z 641.167,A -85,B 0,C 180,E1 21607.552,E2 21607.552} C_VEL
LIN {X 0,Y 226.229,Z 640.374,A -85,B 0,C 180,E1 21619.444,E2 21619.444} C_VEL
LIN {X 0,Y 226.637,Z 641.603,A -85,B 0,C 180,E1 21623.506,E2 21623.506} C_VEL
LIN {X 0,Y 228.574,Z 649.617,A -85,B 0,C 180,E1 21632.621,E2 21632.621} C_VEL
LIN {X 0,Y 231.665,Z 661.142,A -85,B 0,C 180,E1 21640.593,E2 21640.593} C_VEL
LIN {X 0,Y 234.684,Z 675.073,A -85,B 0,C 180,E1 21647.627,E2 21647.627} C_VEL
LIN {X 0,Y 236.232,Z 692.282,A -85,B 0,C 180,E1 21654.33,E2 21654.33} C_VEL
LIN {X 0,Y 235.546,Z 698.319,A -85,B 0,C 180,E1 21656.179,E2 21656.179} C_VEL
LIN {X 0,Y 230.129,Z 707.989,A -85,B 0,C 180,E1 21657.567,E2 21657.567} C_VEL
LIN {X 0,Y 219.894,Z 721.225,A -85,B 0,C 180,E1 21658.939,E2 21658.939} C_VEL
LIN {X 0,Y 209.323,Z 733.606,A -85,B 0,C 180,E1 21660.646,E2 21660.646} C_VEL
LIN {X 0,Y 190.195,Z 758.528,A -85,B 0,C 180,E1 21667.857,E2 21667.857} C_VEL
LIN {X 0,Y 172.847,Z 778.568,A -85,B 0,C 180,E1 21677.389,E2 21677.389} C_VEL
LIN {X 0,Y 160.389,Z 792.531,A -85,B 0,C 180,E1 21688.648,E2 21688.648} C_VEL
LIN {X 0,Y 152.99,Z 801.493,A -85,B 0,C 180,E1 21701.373,E2 21701.373} C_VEL
LIN {X 0,Y 149.804,Z 805.853,A -85,B 0,C 180,E1 21715.104,E2 21715.104} C_VEL
LIN {X 0,Y 151.942,Z 805.73,A -85,B 0,C 180,E1 21727.486,E2 21727.486} C_VEL
LIN {X 0,Y 158.535,Z 801.804,A -85,B 0,C 180,E1 21739.588,E2 21739.588} C_VEL
LIN {X 0,Y 171.201,Z 792.881,A -85,B 0,C 180,E1 21751.807,E2 21751.807} C_VEL
LIN {X 0,Y 190.083,Z 778.28,A -85,B 0,C 180,E1 21762.286,E2 21762.286} C_VEL
LIN {X 0,Y 212.816,Z 758.096,A -85,B 0,C 180,E1 21770.4,E2 21770.4} C_VEL
LIN {X 0,Y 236.507,Z 732.684,A -85,B 0,C 180,E1 21776.373,E2 21776.373} C_VEL
LIN {X 0,Y 251.341,Z 713.505,A -85,B 0,C 180,E1 21779.554,E2 21779.554} C_VEL
LIN {X 0,Y 254.877,Z 705.478,A -85,B 0,C 180,E1 21784.271,E2 21784.271} C_VEL
LIN {X 0,Y 256.17,Z 702.932,A -85,B 0,C 180,E1 21786.793,E2 21786.793} C_VEL
LIN {X 0,Y 256.478,Z 702.789,A -85,B 0,C 180,E1 21790.193,E2 21790.193} C_VEL
LIN {X 0,Y 256.439,Z 706.372,A -85,B 0,C 180,E1 21795.381,E2 21795.381} C_VEL
LIN {X 0,Y 255.363,Z 713.834,A -85,B 0,C 180,E1 21799.889,E2 21799.889} C_VEL
LIN {X 0,Y 253.972,Z 716.528,A -85,B 0,C 180,E1 21800.451,E2 21800.451} C_VEL
LIN {X 0,Y 230.748,Z 747.489,A -85,B 0,C 180,E1 21804.754,E2 21804.754} C_VEL
LIN {X 0,Y 206.665,Z 774.267,A -85,B 0,C 180,E1 21810.892,E2 21810.892} C_VEL
LIN {X 0,Y 183.679,Z 796.794,A -85,B 0,C 180,E1 21819.633,E2 21819.633} C_VEL
LIN {X 0,Y 164.546,Z 814.696,A -85,B 0,C 180,E1 21831.76,E2 21831.76} C_VEL
LIN {X 0,Y 153.216,Z 826.777,A -85,B 0,C 180,E1 21846.804,E2 21846.804} C_VEL
LIN {X 0,Y 150.477,Z 831.473,A -85,B 0,C 180,E1 21858.434,E2 21858.434} C_VEL
LIN {X 0,Y 150.969,Z 832.81,A -85,B 0,C 180,E1 21870.004,E2 21870.004} C_VEL
LIN {X 0,Y 150.58,Z 830.331,A -85,B 0,C 180,E1 21881.566,E2 21881.566} C_VEL
LIN {X 0,Y 154.633,Z 821.89,A -85,B 0,C 180,E1 21896.054,E2 21896.054} C_VEL
LIN {X 0,Y 165.831,Z 807.202,A -85,B 0,C 180,E1 21909.572,E2 21909.572} C_VEL
LIN {X 0,Y 182.14,Z 787.885,A -85,B 0,C 180,E1 21920.033,E2 21920.033} C_VEL
LIN {X 0,Y 200.579,Z 764.717,A -85,B 0,C 180,E1 21927.771,E2 21927.771} C_VEL
LIN {X 0,Y 220.206,Z 736.741,A -85,B 0,C 180,E1 21933.621,E2 21933.621} C_VEL
LIN {X 0,Y 237.805,Z 706.291,A -85,B 0,C 180,E1 21937.731,E2 21937.731} C_VEL
LIN {X 0,Y 236.388,Z 690.806,A -85,B 0,C 180,E1 21942.914,E2 21942.914} C_VEL
LIN {X 0,Y 233.142,Z 674.217,A -85,B 0,C 180,E1 21949.718,E2 21949.718} C_VEL
LIN {X 0,Y 228.943,Z 659.389,A -85,B 0,C 180,E1 21958.002,E2 21958.002} C_VEL
LIN {X 0,Y 226.696,Z 652.048,A -85,B 0,C 180,E1 21963.784,E2 21963.784} C_VEL
LIN {X 0,Y 225.635,Z 648.544,A -85,B 0,C 180,E1 21967.653,E2 21967.653} C_VEL
LIN {X 0,Y 223.274,Z 647.738,A -85,B 0,C 180,E1 21979.712,E2 21979.712} C_VEL
LIN {X 0,Y 223.569,Z 650.7,A -85,B 0,C 180,E1 21985.617,E2 21985.617} C_VEL
LIN {X 0,Y 225.357,Z 657.695,A -85,B 0,C 180,E1 21993.343,E2 21993.343} C_VEL
LIN {X 0,Y 227.935,Z 669.691,A -85,B 0,C 180,E1 22001.401,E2 22001.401} C_VEL
LIN {X 0,Y 230.138,Z 683.889,A -85,B 0,C 180,E1 22008.384,E2 22008.384} C_VEL
LIN {X 0,Y 230.58,Z 699.382,A -85,B 0,C 180,E1 22014.489,E2 22014.489} C_VEL
LIN {X 0,Y 212.546,Z 729.005,A -85,B 0,C 180,E1 22019.609,E2 22019.609} C_VEL
LIN {X 0,Y 209.323,Z 733.606,A -85,B 0,C 180,E1 22020.646,E2 22020.646} C_VEL
LIN {X 0,Y 198.338,Z 745.321,A -85,B 0,C 180,E1 22022.656,E2 22022.656} C_VEL
LIN {X 0,Y 187.114,Z 756.102,A -85,B 0,C 180,E1 22025.059,E2 22025.059} C_VEL
LIN {X 0,Y 168.52,Z 776.805,A -85,B 0,C 180,E1 22034.413,E2 22034.413} C_VEL
LIN {X 0,Y 154.623,Z 791.557,A -85,B 0,C 180,E1 22045.798,E2 22045.798} C_VEL
LIN {X 0,Y 146.323,Z 800.854,A -85,B 0,C 180,E1 22058.309,E2 22058.309} C_VEL
LIN {X 0,Y 142.699,Z 805.096,A -85,B 0,C 180,E1 22068.492,E2 22068.492} C_VEL
LIN {X 0,Y 142.572,Z 806.952,A -85,B 0,C 180,E1 22082.258,E2 22082.258} C_VEL
LIN {X 0,Y 147.854,Z 804.761,A -85,B 0,C 180,E1 22095.59,E2 22095.59} C_VEL
LIN {X 0,Y 158.868,Z 797.99,A -85,B 0,C 180,E1 22108.737,E2 22108.737} C_VEL
LIN {X 0,Y 176.404,Z 785.884,A -85,B 0,C 180,E1 22120.205,E2 22120.205} C_VEL
LIN {X 0,Y 198.283,Z 768.686,A -85,B 0,C 180,E1 22129.016,E2 22129.016} C_VEL
LIN {X 0,Y 222.196,Z 746.294,A -85,B 0,C 180,E1 22135.668,E2 22135.668} C_VEL
LIN {X 0,Y 246.985,Z 717.535,A -85,B 0,C 180,E1 22140.904,E2 22140.904} C_VEL
LIN {X 0,Y 250.463,Z 710.924,A -85,B 0,C 180,E1 22145.213,E2 22145.213} C_VEL
LIN {X 0,Y 251.383,Z 709.304,A -85,B 0,C 180,E1 22146.923,E2 22146.923} C_VEL
LIN {X 0,Y 251.638,Z 710.141,A -85,B 0,C 180,E1 22152.142,E2 22152.142} C_VEL
LIN {X 0,Y 251.279,Z 714.534,A -85,B 0,C 180,E1 22156.6,E2 22156.6} C_VEL
LIN {X 0,Y 250.593,Z 717.62,A -85,B 0,C 180,E1 22158.456,E2 22158.456} C_VEL
LIN {X 0,Y 248.561,Z 721.039,A -85,B 0,C 180,E1 22159.194,E2 22159.194} C_VEL
LIN {X 0,Y 224.743,Z 750.915,A -85,B 0,C 180,E1 22163.493,E2 22163.493} C_VEL
LIN {X 0,Y 198.53,Z 778.274,A -85,B 0,C 180,E1 22170.155,E2 22170.155} C_VEL
LIN {X 0,Y 175.192,Z 799.494,A -85,B 0,C 180,E1 22179.181,E2 22179.181} C_VEL
LIN {X 0,Y 155.999,Z 816.117,A -85,B 0,C 180,E1 22191.798,E2 22191.798} C_VEL
LIN {X 0,Y 145.77,Z 826.155,A -85,B 0,C 180,E1 22205.544,E2 22205.544} C_VEL
LIN {X 0,Y 142.614,Z 830.79,A -85,B 0,C 180,E1 22217.787,E2 22217.787} C_VEL
LIN {X 0,Y 143.089,Z 832.084,A -85,B 0,C 180,E1 22230.005,E2 22230.005} C_VEL
LIN {X 0,Y 142.739,Z 829.493,A -85,B 0,C 180,E1 22242.211,E2 22242.211} C_VEL
LIN {X 0,Y 147.351,Z 820.921,A -85,B 0,C 180,E1 22257.446,E2 22257.446} C_VEL
LIN {X 0,Y 159.541,Z 806.05,A -85,B 0,C 180,E1 22271.465,E2 22271.465} C_VEL
LIN {X 0,Y 176.597,Z 786.928,A -85,B 0,C 180,E1 22281.925,E2 22281.925} C_VEL
LIN {X 0,Y 195.97,Z 763.494,A -85,B 0,C 180,E1 22289.724,E2 22289.724} C_VEL
LIN {X 0,Y 216.524,Z 734.927,A -85,B 0,C 180,E1 22295.562,E2 22295.562} C_VEL
LIN {X 0,Y 232.38,Z 708.226,A -85,B 0,C 180,E1 22299.171,E2 22299.171} C_VEL
LIN {X 0,Y 230.063,Z 688.016,A -85,B 0,C 180,E1 22306.82,E2 22306.82} C_VEL
LIN {X 0,Y 226.834,Z 672.837,A -85,B 0,C 180,E1 22314.243,E2 22314.243} C_VEL
LIN {X 0,Y 223.666,Z 660.343,A -85,B 0,C 180,E1 22322.869,E2 22322.869} C_VEL
LIN {X 0,Y 222.333,Z 655.765,A -85,B 0,C 180,E1 22327.767,E2 22327.767} C_VEL
LIN {X 0,Y 220.121,Z 654.7,A -85,B 0,C 180,E1 22336.3,E2 22336.3} C_VEL
LIN {X 0,Y 220.215,Z 656.907,A -85,B 0,C 180,E1 22344.235,E2 22344.235} C_VEL
LIN {X 0,Y 221.564,Z 664.481,A -85,B 0,C 180,E1 22352.968,E2 22352.968} C_VEL
LIN {X 0,Y 223.608,Z 676.388,A -85,B 0,C 180,E1 22361.175,E2 22361.175} C_VEL
LIN {X 0,Y 225.048,Z 690.944,A -85,B 0,C 180,E1 22368.465,E2 22368.465} C_VEL
LIN {X 0,Y 224.683,Z 703.433,A -85,B 0,C 180,E1 22373.408,E2 22373.408} C_VEL
LIN {X 0,Y 205.784,Z 732.344,A -85,B 0,C 180,E1 22378.498,E2 22378.498} C_VEL
LIN {X 0,Y 187.114,Z 756.102,A -85,B 0,C 180,E1 22385.059,E2 22385.059} C_VEL
LIN {X 0,Y 175.898,Z 766.069,A -85,B 0,C 180,E1 22387.944,E2 22387.944} C_VEL
LIN {X 0,Y 164.672,Z 775.049,A -85,B 0,C 180,E1 22391.345,E2 22391.345} C_VEL
LIN {X 0,Y 149.242,Z 790.505,A -85,B 0,C 180,E1 22402.733,E2 22402.733} C_VEL
LIN {X 0,Y 139.314,Z 800.813,A -85,B 0,C 180,E1 22416.214,E2 22416.214} C_VEL
LIN {X 0,Y 134.552,Z 806.187,A -85,B 0,C 180,E1 22429.656,E2 22429.656} C_VEL
LIN {X 0,Y 135.024,Z 807.678,A -85,B 0,C 180,E1 22443.967,E2 22443.967} C_VEL
LIN {X 0,Y 141.464,Z 805.101,A -85,B 0,C 180,E1 22458.298,E2 22458.298} C_VEL
LIN {X 0,Y 154.087,Z 797.928,A -85,B 0,C 180,E1 22471.802,E2 22471.802} C_VEL
LIN {X 0,Y 173.358,Z 785.425,A -85,B 0,C 180,E1 22483.224,E2 22483.224} C_VEL
LIN {X 0,Y 198.005,Z 766.777,A -85,B 0,C 180,E1 22492.174,E2 22492.174} C_VEL
LIN {X 0,Y 223.964,Z 742.692,A -85,B 0,C 180,E1 22498.572,E2 22498.572} C_VEL
LIN {X 0,Y 241.564,Z 722.976,A -85,B 0,C 180,E1 22501.902,E2 22501.902} C_VEL
LIN {X 0,Y 244.617,Z 718.283,A -85,B 0,C 180,E1 22504.451,E2 22504.451} C_VEL
LIN {X 0,Y 246.4,Z 715.534,A -85,B 0,C 180,E1 22507.063,E2 22507.063} C_VEL
LIN {X 0,Y 246.744,Z 716.237,A -85,B 0,C 180,E1 22511.912,E2 22511.912} C_VEL
LIN {X 0,Y 246.378,Z 719.164,A -85,B 0,C 180,E1 22515.356,E2 22515.356} C_VEL
LIN {X 0,Y 245.28,Z 722.845,A -85,B 0,C 180,E1 22517.579,E2 22517.579} C_VEL
LIN {X 0,Y 220.508,Z 752.502,A -85,B 0,C 180,E1 22521.823,E2 22521.823} C_VEL
LIN {X 0,Y 193.597,Z 779.054,A -85,B 0,C 180,E1 22528.367,E2 22528.367} C_VEL
LIN {X 0,Y 168.385,Z 800.566,A -85,B 0,C 180,E1 22537.865,E2 22537.865} C_VEL
LIN {X 0,Y 149.444,Z 815.782,A -85,B 0,C 180,E1 22550.017,E2 22550.017} C_VEL
LIN {X 0,Y 138.374,Z 825.539,A -85,B 0,C 180,E1 22564.143,E2 22564.143} C_VEL
LIN {X 0,Y 134.764,Z 830.111,A -85,B 0,C 180,E1 22577.064,E2 22577.064} C_VEL
LIN {X 0,Y 135.207,Z 831.354,A -85,B 0,C 180,E1 22590.005,E2 22590.005} C_VEL
LIN {X 0,Y 134.911,Z 828.647,A -85,B 0,C 180,E1 22602.932,E2 22602.932} C_VEL
LIN {X 0,Y 139.961,Z 820.147,A -85,B 0,C 180,E1 22618.705,E2 22618.705} C_VEL
LIN {X 0,Y 152.34,Z 806.069,A -85,B 0,C 180,E1 22632.659,E2 22632.659} C_VEL
LIN {X 0,Y 170.56,Z 786.694,A -85,B 0,C 180,E1 22643.618,E2 22643.618} C_VEL
LIN {X 0,Y 191.64,Z 762.188,A -85,B 0,C 180,E1 22651.771,E2 22651.771} C_VEL
LIN {X 0,Y 213.231,Z 732.944,A -85,B 0,C 180,E1 22657.589,E2 22657.589} C_VEL
LIN {X 0,Y 226.615,Z 711.118,A -85,B 0,C 180,E1 22660.523,E2 22660.523} C_VEL
LIN {X 0,Y 224.928,Z 692.641,A -85,B 0,C 180,E1 22667.868,E2 22667.868} C_VEL
LIN {X 0,Y 222.387,Z 678.557,A -85,B 0,C 180,E1 22675.103,E2 22675.103} C_VEL
LIN {X 0,Y 220.013,Z 667.51,A -85,B 0,C 180,E1 22682.915,E2 22682.915} C_VEL
LIN {X 0,Y 218.9,Z 662.912,A -85,B 0,C 180,E1 22687.89,E2 22687.89} C_VEL
LIN {X 0,Y 216.782,Z 661.809,A -85,B 0,C 180,E1 22696.129,E2 22696.129} C_VEL
LIN {X 0,Y 216.556,Z 663.447,A -85,B 0,C 180,E1 22702.926,E2 22702.926} C_VEL
LIN {X 0,Y 217.325,Z 669.634,A -85,B 0,C 180,E1 22711.127,E2 22711.127} C_VEL
LIN {X 0,Y 218.64,Z 679.993,A -85,B 0,C 180,E1 22719.063,E2 22719.063} C_VEL
LIN {X 0,Y 219.788,Z 693.74,A -85,B 0,C 180,E1 22726.636,E2 22726.636} C_VEL
LIN {X 0,Y 219.402,Z 705.457,A -85,B 0,C 180,E1 22731.753,E2 22731.753} C_VEL
LIN {X 0,Y 200.407,Z 733.823,A -85,B 0,C 180,E1 22736.909,E2 22736.909} C_VEL
LIN {X 0,Y 180.142,Z 758.502,A -85,B 0,C 180,E1 22743.906,E2 22743.906} C_VEL
LIN {X 0,Y 164.672,Z 775.049,A -85,B 0,C 180,E1 22751.345,E2 22751.345} C_VEL
LIN {X 0,Y 153.782,Z 783.054,A -85,B 0,C 180,E1 22755.394,E2 22755.394} C_VEL
LIN {X 0,Y 143.487,Z 790.08,A -85,B 0,C 180,E1 22760.159,E2 22760.159} C_VEL
LIN {X 0,Y 132.804,Z 800.364,A -85,B 0,C 180,E1 22773.252,E2 22773.252} C_VEL
LIN {X 0,Y 126.923,Z 806.501,A -85,B 0,C 180,E1 22788.21,E2 22788.21} C_VEL
LIN {X 0,Y 127.684,Z 808.403,A -85,B 0,C 180,E1 22806.216,E2 22806.216} C_VEL
LIN {X 0,Y 135.349,Z 805.459,A -85,B 0,C 180,E1 22821.293,E2 22821.293} C_VEL
LIN {X 0,Y 152.123,Z 796.552,A -85,B 0,C 180,E1 22836.68,E2 22836.68} C_VEL
LIN {X 0,Y 173.418,Z 783.258,A -85,B 0,C 180,E1 22847.351,E2 22847.351} C_VEL
LIN {X 0,Y 199.848,Z 763.453,A -85,B 0,C 180,E1 22855.707,E2 22855.707} C_VEL
LIN {X 0,Y 226.412,Z 738.882,A -85,B 0,C 180,E1 22861.443,E2 22861.443} C_VEL
LIN {X 0,Y 238.256,Z 725.798,A -85,B 0,C 180,E1 22863.661,E2 22863.661} C_VEL
LIN {X 0,Y 241.298,Z 721.693,A -85,B 0,C 180,E1 22867.213,E2 22867.213} C_VEL
LIN {X 0,Y 241.645,Z 722.559,A -85,B 0,C 180,E1 22872.167,E2 22872.167} C_VEL
LIN {X 0,Y 240.841,Z 726.123,A -85,B 0,C 180,E1 22875.859,E2 22875.859} C_VEL
LIN {X 0,Y 234.679,Z 733.956,A -85,B 0,C 180,E1 22877.001,E2 22877.001} C_VEL
LIN {X 0,Y 207.408,Z 763.057,A -85,B 0,C 180,E1 22881.939,E2 22881.939} C_VEL
LIN {X 0,Y 180.971,Z 786.515,A -85,B 0,C 180,E1 22888.899,E2 22888.899} C_VEL
LIN {X 0,Y 156.035,Z 805.858,A -85,B 0,C 180,E1 22899.321,E2 22899.321} C_VEL
LIN {X 0,Y 137.879,Z 819.359,A -85,B 0,C 180,E1 22912.997,E2 22912.997} C_VEL
LIN {X 0,Y 128.002,Z 828.021,A -85,B 0,C 180,E1 22930.713,E2 22930.713} C_VEL
LIN {X 0,Y 126.571,Z 830.446,A -85,B 0,C 180,E1 22943.158,E2 22943.158} C_VEL
LIN {X 0,Y 127.319,Z 830.624,A -85,B 0,C 180,E1 22950.005,E2 22950.005} C_VEL
LIN {X 0,Y 127.103,Z 827.792,A -85,B 0,C 180,E1 22963.741,E2 22963.741} C_VEL
LIN {X 0,Y 132.712,Z 819.296,A -85,B 0,C 180,E1 22980.203,E2 22980.203} C_VEL
LIN {X 0,Y 146.394,Z 804.853,A -85,B 0,C 180,E1 22994.868,E2 22994.868} C_VEL
LIN {X 0,Y 166.1,Z 784.89,A -85,B 0,C 180,E1 23006.11,E2 23006.11} C_VEL
LIN {X 0,Y 187.824,Z 760.484,A -85,B 0,C 180,E1 23014.022,E2 23014.022} C_VEL
LIN {X 0,Y 210.168,Z 730.869,A -85,B 0,C 180,E1 23019.688,E2 23019.688} C_VEL
LIN {X 0,Y 220.8,Z 713.607,A -85,B 0,C 180,E1 23022.061,E2 23022.061} C_VEL
LIN {X 0,Y 219.663,Z 695.944,A -85,B 0,C 180,E1 23029.58,E2 23029.58} C_VEL
LIN {X 0,Y 217.368,Z 681.116,A -85,B 0,C 180,E1 23037.978,E2 23037.978} C_VEL
LIN {X 0,Y 216.018,Z 673.536,A -85,B 0,C 180,E1 23043.971,E2 23043.971} C_VEL
LIN {X 0,Y 215.256,Z 669.973,A -85,B 0,C 180,E1 23048.024,E2 23048.024} C_VEL
LIN {X 0,Y 213.211,Z 668.896,A -85,B 0,C 180,E1 23056.406,E2 23056.406} C_VEL
LIN {X 0,Y 212.9,Z 670.468,A -85,B 0,C 180,E1 23062.857,E2 23062.857} C_VEL
LIN {X 0,Y 213.465,Z 677.502,A -85,B 0,C 180,E1 23071.967,E2 23071.967} C_VEL
LIN {X 0,Y 214.322,Z 689.133,A -85,B 0,C 180,E1 23080.521,E2 23080.521} C_VEL
LIN {X 0,Y 214.376,Z 702.794,A -85,B 0,C 180,E1 23087.744,E2 23087.744} C_VEL
LIN {X 0,Y 213.742,Z 709.163,A -85,B 0,C 180,E1 23090.547,E2 23090.547} C_VEL
LIN {X 0,Y 192.522,Z 738.788,A -85,B 0,C 180,E1 23096.046,E2 23096.046} C_VEL
LIN {X 0,Y 170.648,Z 763.628,A -85,B 0,C 180,E1 23103.755,E2 23103.755} C_VEL
LIN {X 0,Y 151.396,Z 782.654,A -85,B 0,C 180,E1 23114.02,E2 23114.02} C_VEL
LIN {X 0,Y 143.487,Z 790.08,A -85,B 0,C 180,E1 23120.159,E2 23120.159} C_VEL
LIN {X 0,Y 133.917,Z 796.04,A -85,B 0,C 180,E1 23125.72,E2 23125.72} C_VEL
LIN {X 0,Y 125.326,Z 800.985,A -85,B 0,C 180,E1 23132.154,E2 23132.154} C_VEL
LIN {X 0,Y 119.939,Z 806.261,A -85,B 0,C 180,E1 23144.568,E2 23144.568} C_VEL
LIN {X 0,Y 118.57,Z 809.086,A -85,B 0,C 180,E1 23160.595,E2 23160.595} C_VEL
LIN {X 0,Y 124.208,Z 807.919,A -85,B 0,C 180,E1 23176.79,E2 23176.79} C_VEL
LIN {X 0,Y 136.897,Z 802.404,A -85,B 0,C 180,E1 23191.855,E2 23191.855} C_VEL
LIN {X 0,Y 156.67,Z 791.886,A -85,B 0,C 180,E1 23204.388,E2 23204.388} C_VEL
LIN {X 0,Y 182.107,Z 775.667,A -85,B 0,C 180,E1 23213.882,E2 23213.882} C_VEL
LIN {X 0,Y 209.871,Z 753.796,A -85,B 0,C 180,E1 23220.681,E2 23220.681} C_VEL
LIN {X 0,Y 233.985,Z 730.081,A -85,B 0,C 180,E1 23225.117,E2 23225.117} C_VEL
LIN {X 0,Y 235.954,Z 727.664,A -85,B 0,C 180,E1 23227.378,E2 23227.378} C_VEL
LIN {X 0,Y 236.43,Z 727.892,A -85,B 0,C 180,E1 23231.067,E2 23231.067} C_VEL
LIN {X 0,Y 235.94,Z 730.272,A -85,B 0,C 180,E1 23234.329,E2 23234.329} C_VEL
LIN {X 0,Y 233.375,Z 733.587,A -85,B 0,C 180,E1 23235.018,E2 23235.018} C_VEL
LIN {X 0,Y 206.133,Z 761.797,A -85,B 0,C 180,E1 23239.53,E2 23239.53} C_VEL
LIN {X 0,Y 178.6,Z 785.311,A -85,B 0,C 180,E1 23246.148,E2 23246.148} C_VEL
LIN {X 0,Y 153.35,Z 803.917,A -85,B 0,C 180,E1 23255.737,E2 23255.737} C_VEL
LIN {X 0,Y 132.993,Z 817.777,A -85,B 0,C 180,E1 23269.282,E2 23269.282} C_VEL
LIN {X 0,Y 120.827,Z 826.95,A -85,B 0,C 180,E1 23288.002,E2 23288.002} C_VEL
LIN {X 0,Y 118.66,Z 829.744,A -85,B 0,C 180,E1 23302.699,E2 23302.699} C_VEL
LIN {X 0,Y 119.428,Z 829.892,A -85,B 0,C 180,E1 23310.005,E2 23310.005} C_VEL
LIN {X 0,Y 119.325,Z 826.931,A -85,B 0,C 180,E1 23324.656,E2 23324.656} C_VEL
LIN {X 0,Y 125.193,Z 818.859,A -85,B 0,C 180,E1 23341.25,E2 23341.25} C_VEL
LIN {X 0,Y 139.658,Z 804.604,A -85,B 0,C 180,E1 23356.515,E2 23356.515} C_VEL
LIN {X 0,Y 160.234,Z 784.838,A -85,B 0,C 180,E1 23367.957,E2 23367.957} C_VEL
LIN {X 0,Y 182.128,Z 761.286,A -85,B 0,C 180,E1 23375.708,E2 23375.708} C_VEL
LIN {X 0,Y 205.06,Z 732.067,A -85,B 0,C 180,E1 23381.341,E2 23381.341} C_VEL
LIN {X 0,Y 215.094,Z 716.79,A -85,B 0,C 180,E1 23383.41,E2 23383.41} C_VEL
LIN {X 0,Y 214.508,Z 700.216,A -85,B 0,C 180,E1 23390.857,E2 23390.857} C_VEL
LIN {X 0,Y 212.889,Z 686.752,A -85,B 0,C 180,E1 23398.951,E2 23398.951} C_VEL
LIN {X 0,Y 211.622,Z 678.634,A -85,B 0,C 180,E1 23406.102,E2 23406.102} C_VEL
LIN {X 0,Y 211.372,Z 676.891,A -85,B 0,C 180,E1 23408.173,E2 23408.173} C_VEL
LIN {X 0,Y 209.339,Z 675.883,A -85,B 0,C 180,E1 23416.719,E2 23416.719} C_VEL
LIN {X 0,Y 208.993,Z 677.68,A -85,B 0,C 180,E1 23423.309,E2 23423.309} C_VEL
LIN {X 0,Y 209.151,Z 683.848,A -85,B 0,C 180,E1 23431.489,E2 23431.489} C_VEL
LIN {X 0,Y 209.482,Z 695.653,A -85,B 0,C 180,E1 23440.358,E2 23440.358} C_VEL
LIN {X 0,Y 208.765,Z 708.95,A -85,B 0,C 180,E1 23447.566,E2 23447.566} C_VEL
LIN {X 0,Y 207.705,Z 713.111,A -85,B 0,C 180,E1 23449.162,E2 23449.162} C_VEL
LIN {X 0,Y 186.047,Z 741.786,A -85,B 0,C 180,E1 23454.692,E2 23454.692} C_VEL
LIN {X 0,Y 164.76,Z 764.822,A -85,B 0,C 180,E1 23462.001,E2 23462.001} C_VEL
LIN {X 0,Y 145.557,Z 782.914,A -85,B 0,C 180,E1 23471.875,E2 23471.875} C_VEL
LIN {X 0,Y 129.742,Z 796.978,A -85,B 0,C 180,E1 23485.832,E2 23485.832} C_VEL
LIN {X 0,Y 125.326,Z 800.985,A -85,B 0,C 180,E1 23492.154,E2 23492.154} C_VEL
LIN {X 0,Y 119.97,Z 804.019,A -85,B 0,C 180,E1 23497.566,E2 23497.566} C_VEL
LIN {X 0,Y 111.179,Z 807.794,A -85,B 0,C 180,E1 23507.473,E2 23507.473} C_VEL
LIN {X 0,Y 111.632,Z 809.894,A -85,B 0,C 180,E1 23525.928,E2 23525.928} C_VEL
LIN {X 0,Y 120.969,Z 807.357,A -85,B 0,C 180,E1 23544.149,E2 23544.149} C_VEL
LIN {X 0,Y 138.868,Z 799.637,A -85,B 0,C 180,E1 23559.848,E2 23559.848} C_VEL
LIN {X 0,Y 164.539,Z 785.879,A -85,B 0,C 180,E1 23571.753,E2 23571.753} C_VEL
LIN {X 0,Y 193.244,Z 766.5,A -85,B 0,C 180,E1 23579.815,E2 23579.815} C_VEL
LIN {X 0,Y 222.051,Z 741.935,A -85,B 0,C 180,E1 23585.265,E2 23585.265} C_VEL
LIN {X 0,Y 229.505,Z 734.487,A -85,B 0,C 180,E1 23586.544,E2 23586.544} C_VEL
LIN {X 0,Y 230.449,Z 733.541,A -85,B 0,C 180,E1 23587.555,E2 23587.555} C_VEL
LIN {X 0,Y 230.75,Z 734.487,A -85,B 0,C 180,E1 23592.188,E2 23592.188} C_VEL
LIN {X 0,Y 230.637,Z 734.98,A -85,B 0,C 180,E1 23592.942,E2 23592.942} C_VEL
LIN {X 0,Y 222.712,Z 743.667,A -85,B 0,C 180,E1 23594.305,E2 23594.305} C_VEL
LIN {X 0,Y 193.793,Z 770.571,A -85,B 0,C 180,E1 23599.31,E2 23599.31} C_VEL
LIN {X 0,Y 164.599,Z 792.898,A -85,B 0,C 180,E1 23606.973,E2 23606.973} C_VEL
LIN {X 0,Y 138.919,Z 809.806,A -85,B 0,C 180,E1 23618.185,E2 23618.185} C_VEL
LIN {X 0,Y 119.705,Z 821.809,A -85,B 0,C 180,E1 23634.562,E2 23634.562} C_VEL
LIN {X 0,Y 111.367,Z 828.093,A -85,B 0,C 180,E1 23654.282,E2 23654.282} C_VEL
LIN {X 0,Y 111.531,Z 829.156,A -85,B 0,C 180,E1 23670.006,E2 23670.006} C_VEL
LIN {X 0,Y 111.572,Z 826.059,A -85,B 0,C 180,E1 23685.7,E2 23685.7} C_VEL
LIN {X 0,Y 118.276,Z 817.83,A -85,B 0,C 180,E1 23703.307,E2 23703.307} C_VEL
LIN {X 0,Y 134.565,Z 802.98,A -85,B 0,C 180,E1 23719.368,E2 23719.368} C_VEL
LIN {X 0,Y 155.98,Z 783.36,A -85,B 0,C 180,E1 23730.548,E2 23730.548} C_VEL
LIN {X 0,Y 178.87,Z 759.514,A -85,B 0,C 180,E1 23738.135,E2 23738.135} C_VEL
LIN {X 0,Y 202.882,Z 729.411,A -85,B 0,C 180,E1 23743.636,E2 23743.636} C_VEL
LIN {X 0,Y 209.454,Z 719.389,A -85,B 0,C 180,E1 23745.062,E2 23745.062} C_VEL
LIN {X 0,Y 209.301,Z 703.475,A -85,B 0,C 180,E1 23752.719,E2 23752.719} C_VEL
LIN {X 0,Y 208.191,Z 691.132,A -85,B 0,C 180,E1 23760.869,E2 23760.869} C_VEL
LIN {X 0,Y 207.368,Z 683.721,A -85,B 0,C 180,E1 23768.331,E2 23768.331} C_VEL
LIN {X 0,Y 205.328,Z 682.797,A -85,B 0,C 180,E1 23777.164,E2 23777.164} C_VEL
LIN {X 0,Y 204.808,Z 684.838,A -85,B 0,C 180,E1 23783.861,E2 23783.861} C_VEL
LIN {X 0,Y 204.676,Z 691.601,A -85,B 0,C 180,E1 23792.337,E2 23792.337} C_VEL
LIN {X 0,Y 204.312,Z 702.832,A -85,B 0,C 180,E1 23800.685,E2 23800.685} C_VEL
LIN {X 0,Y 203.141,Z 714.43,A -85,B 0,C 180,E1 23807.077,E2 23807.077} C_VEL
LIN {X 0,Y 198.76,Z 721.039,A -85,B 0,C 180,E1 23808.366,E2 23808.366} C_VEL
LIN {X 0,Y 175.566,Z 749.277,A -85,B 0,C 180,E1 23814.413,E2 23814.413} C_VEL
LIN {X 0,Y 152.914,Z 771.774,A -85,B 0,C 180,E1 23822.781,E2 23822.781} C_VEL
LIN {X 0,Y 132.624,Z 789.325,A -85,B 0,C 180,E1 23834.68,E2 23834.68} C_VEL
LIN {X 0,Y 118.492,Z 801.145,A -85,B 0,C 180,E1 23849.995,E2 23849.995} C_VEL
LIN {X 0,Y 111.648,Z 807.337,A -85,B 0,C 180,E1 23865.677,E2 23865.677} C_VEL
LIN {X 0,Y 111.179,Z 807.794,A -85,B 0,C 180,E1 23867.473,E2 23867.473} C_VEL
LIN {X 0,Y 106.441,Z 809.868,A -85,B 0,C 180,E1 23876.295,E2 23876.295} C_VEL
LIN {X 0,Y 103.658,Z 810.624,A -85,B 0,C 180,E1 23885.799,E2 23885.799} C_VEL
LIN {X 0,Y 112.28,Z 808.883,A -85,B 0,C 180,E1 23903.734,E2 23903.734} C_VEL
LIN {X 0,Y 129.178,Z 802.612,A -85,B 0,C 180,E1 23919.55,E2 23919.55} C_VEL
LIN {X 0,Y 155.542,Z 789.877,A -85,B 0,C 180,E1 23932.435,E2 23932.435} C_VEL
LIN {X 0,Y 184.372,Z 772.257,A -85,B 0,C 180,E1 23940.658,E2 23940.658} C_VEL
LIN {X 0,Y 214.048,Z 749.187,A -85,B 0,C 180,E1 23946.273,E2 23946.273} C_VEL
LIN {X 0,Y 224.055,Z 740.049,A -85,B 0,C 180,E1 23947.772,E2 23947.772} C_VEL
LIN {X 0,Y 225.259,Z 739.807,A -85,B 0,C 180,E1 23951.624,E2 23951.624} C_VEL
LIN {X 0,Y 193.941,Z 768.629,A -85,B 0,C 180,E1 23956.52,E2 23956.52} C_VEL
LIN {X 0,Y 164.39,Z 790.578,A -85,B 0,C 180,E1 23963.383,E2 23963.383} C_VEL
LIN {X 0,Y 135.185,Z 808.766,A -85,B 0,C 180,E1 23974.783,E2 23974.783} C_VEL
LIN {X 0,Y 113.194,Z 821.24,A -85,B 0,C 180,E1 23992.088,E2 23992.088} C_VEL
LIN {X 0,Y 103.634,Z 827.427,A -85,B 0,C 180,E1 24013.075,E2 24013.075} C_VEL
LIN {X 0,Y 103.623,Z 828.389,A -85,B 0,C 180,E1 24030.006,E2 24030.006} C_VEL
LIN {X 0,Y 103.842,Z 825.178,A -85,B 0,C 180,E1 24046.903,E2 24046.903} C_VEL
LIN {X 0,Y 111.518,Z 816.765,A -85,B 0,C 180,E1 24065.627,E2 24065.627} C_VEL
LIN {X 0,Y 129.182,Z 801.851,A -85,B 0,C 180,E1 24082.052,E2 24082.052} C_VEL
LIN {X 0,Y 152.093,Z 781.856,A -85,B 0,C 180,E1 24093.256,E2 24093.256} C_VEL
LIN {X 0,Y 177.537,Z 755.984,A -85,B 0,C 180,E1 24101.024,E2 24101.024} C_VEL
LIN {X 0,Y 202.067,Z 725.144,A -85,B 0,C 180,E1 24106.139,E2 24106.139} C_VEL
LIN {X 0,Y 203.865,Z 721.204,A -85,B 0,C 180,E1 24107.137,E2 24107.137} C_VEL
LIN {X 0,Y 204.123,Z 706.904,A -85,B 0,C 180,E1 24114.664,E2 24114.664} C_VEL
LIN {X 0,Y 203.529,Z 695.223,A -85,B 0,C 180,E1 24123.152,E2 24123.152} C_VEL
LIN {X 0,Y 203.124,Z 690.394,A -85,B 0,C 180,E1 24128.507,E2 24128.507} C_VEL
LIN {X 0,Y 201.131,Z 689.594,A -85,B 0,C 180,E1 24137.422,E2 24137.422} C_VEL
LIN {X 0,Y 200.404,Z 692.422,A -85,B 0,C 180,E1 24145.36,E2 24145.36} C_VEL
LIN {X 0,Y 199.965,Z 699.058,A -85,B 0,C 180,E1 24153.027,E2 24153.027} C_VEL
LIN {X 0,Y 199.03,Z 709.327,A -85,B 0,C 180,E1 24160.691,E2 24160.691} C_VEL
LIN {X 0,Y 197.731,Z 717.723,A -85,B 0,C 180,E1 24165.538,E2 24165.538} C_VEL
LIN {X 0,Y 175.109,Z 745.672,A -85,B 0,C 180,E1 24171.164,E2 24171.164} C_VEL
LIN {X 0,Y 150.912,Z 769.551,A -85,B 0,C 180,E1 24179.167,E2 24179.167} C_VEL
LIN {X 0,Y 128.401,Z 788.334,A -85,B 0,C 180,E1 24191.075,E2 24191.075} C_VEL
LIN {X 0,Y 112.596,Z 800.653,A -85,B 0,C 180,E1 24206.452,E2 24206.452} C_VEL
LIN {X 0,Y 104.598,Z 807.307,A -85,B 0,C 180,E1 24222.491,E2 24222.491} C_VEL
LIN {X 0,Y 102.496,Z 810.228,A -85,B 0,C 180,E1 24238.125,E2 24238.125} C_VEL
LIN {X 0,Y 103.658,Z 810.624,A -85,B 0,C 180,E1 24245.799,E2 24245.799} C_VEL
LIN {X 0,Y 103.102,Z 810.668,A -85,B 0,C 180,E1 24255.522,E2 24255.522} C_VEL
LIN {X 0,Y 104.915,Z 809.872,A -85,B 0,C 180,E1 24265.181,E2 24265.181} C_VEL
LIN {X 0,Y 125.879,Z 802.774,A -85,B 0,C 180,E1 24283.523,E2 24283.523} C_VEL
LIN {X 0,Y 153.78,Z 790.042,A -85,B 0,C 180,E1 24295.682,E2 24295.682} C_VEL
LIN {X 0,Y 185.564,Z 771.18,A -85,B 0,C 180,E1 24303.748,E2 24303.748} C_VEL
LIN {X 0,Y 215.851,Z 747.841,A -85,B 0,C 180,E1 24308.8,E2 24308.8} C_VEL
LIN {X 0,Y 218.674,Z 745.329,A -85,B 0,C 180,E1 24309.448,E2 24309.448} C_VEL
LIN {X 0,Y 218.874,Z 745.303,A -85,B 0,C 180,E1 24310.069,E2 24310.069} C_VEL
LIN {X 0,Y 195.971,Z 765.647,A -85,B 0,C 180,E1 24313.521,E2 24313.521} C_VEL
LIN {X 0,Y 164.422,Z 788.566,A -85,B 0,C 180,E1 24319.91,E2 24319.91} C_VEL
LIN {X 0,Y 133.785,Z 806.786,A -85,B 0,C 180,E1 24330.377,E2 24330.377} C_VEL
LIN {X 0,Y 109.536,Z 819.326,A -85,B 0,C 180,E1 24346.471,E2 24346.471} C_VEL
LIN {X 0,Y 98.624,Z 825.071,A -85,B 0,C 180,E1 24362.683,E2 24362.683} C_VEL
LIN {X 0,Y 94.954,Z 827.635,A -85,B 0,C 180,E1 24380.863,E2 24380.863} C_VEL
LIN {X 0,Y 95.717,Z 827.606,A -85,B 0,C 180,E1 24390.007,E2 24390.007} C_VEL
LIN {X 0,Y 96.54,Z 823.775,A -85,B 0,C 180,E1 24410.126,E2 24410.126} C_VEL
LIN {X 0,Y 107.108,Z 813.978,A -85,B 0,C 180,E1 24430.959,E2 24430.959} C_VEL
LIN {X 0,Y 128.081,Z 797.552,A -85,B 0,C 180,E1 24447.251,E2 24447.251} C_VEL
LIN {X 0,Y 152.985,Z 776.192,A -85,B 0,C 180,E1 24457.638,E2 24457.638} C_VEL
LIN {X 0,Y 178.066,Z 750.575,A -85,B 0,C 180,E1 24464.263,E2 24464.263} C_VEL
LIN {X 0,Y 197.58,Z 726.409,A -85,B 0,C 180,E1 24467.996,E2 24467.996} C_VEL
LIN {X 0,Y 198.738,Z 719.412,A -85,B 0,C 180,E1 24471.231,E2 24471.231} C_VEL
LIN {X 0,Y 198.904,Z 707.247,A -85,B 0,C 180,E1 24478.877,E2 24478.877} C_VEL
LIN {X 0,Y 198.749,Z 698.673,A -85,B 0,C 180,E1 24486.502,E2 24486.502} C_VEL
LIN {X 0,Y 198.606,Z 696.908,A -85,B 0,C 180,E1 24488.959,E2 24488.959} C_VEL
LIN {X 0,Y 196.672,Z 696.287,A -85,B 0,C 180,E1 24497.83,E2 24497.83} C_VEL
LIN {X 0,Y 195.829,Z 699.472,A -85,B 0,C 180,E1 24505.996,E2 24505.996} C_VEL
LIN {X 0,Y 195.052,Z 705.261,A -85,B 0,C 180,E1 24512.737,E2 24512.737} C_VEL
LIN {X 0,Y 193.643,Z 715.095,A -85,B 0,C 180,E1 24520.267,E2 24520.267} C_VEL
LIN {X 0,Y 192.419,Z 721.12,A -85,B 0,C 180,E1 24523.964,E2 24523.964} C_VEL
LIN {X 0,Y 168.709,Z 748.853,A -85,B 0,C 180,E1 24529.549,E2 24529.549} C_VEL
LIN {X 0,Y 144.145,Z 771.797,A -85,B 0,C 180,E1 24537.548,E2 24537.548} C_VEL
LIN {X 0,Y 120.785,Z 790.089,A -85,B 0,C 180,E1 24549.832,E2 24549.832} C_VEL
LIN {X 0,Y 104.148,Z 802.233,A -85,B 0,C 180,E1 24566.558,E2 24566.558} C_VEL
LIN {X 0,Y 96.282,Z 808.392,A -85,B 0,C 180,E1 24583.459,E2 24583.459} C_VEL
LIN {X 0,Y 95.791,Z 811.273,A -85,B 0,C 180,E1 24606.474,E2 24606.474} C_VEL
LIN {X 0,Y 104.915,Z 809.872,A -85,B 0,C 180,E1 24625.181,E2 24625.181} C_VEL
LIN {X 0,Y 108.818,Z 808.296,A -85,B 0,C 180,E1 24634.318,E2 24634.318} C_VEL
LIN {X 0,Y 114.877,Z 805.924,A -85,B 0,C 180,E1 24642.702,E2 24642.702} C_VEL
LIN {X 0,Y 142.644,Z 794.956,A -85,B 0,C 180,E1 24655.893,E2 24655.893} C_VEL
LIN {X 0,Y 173.309,Z 778.9,A -85,B 0,C 180,E1 24664.104,E2 24664.104} C_VEL
LIN {X 0,Y 203.885,Z 758.112,A -85,B 0,C 180,E1 24669.402,E2 24669.402} C_VEL
LIN {X 0,Y 201.833,Z 759.909,A -85,B 0,C 180,E1 24670.185,E2 24670.185} C_VEL
LIN {X 0,Y 169.251,Z 783.8,A -85,B 0,C 180,E1 24675.554,E2 24675.554} C_VEL
LIN {X 0,Y 136.778,Z 802.891,A -85,B 0,C 180,E1 24684.48,E2 24684.48} C_VEL
LIN {X 0,Y 107.143,Z 817.351,A -85,B 0,C 180,E1 24700.375,E2 24700.375} C_VEL
LIN {X 0,Y 91.459,Z 824.459,A -85,B 0,C 180,E1 24720.34,E2 24720.34} C_VEL
LIN {X 0,Y 87.077,Z 826.896,A -85,B 0,C 180,E1 24740.028,E2 24740.028} C_VEL
LIN {X 0,Y 87.802,Z 826.818,A -85,B 0,C 180,E1 24750.007,E2 24750.007} C_VEL
LIN {X 0,Y 88.576,Z 823.394,A -85,B 0,C 180,E1 24769.929,E2 24769.929} C_VEL
LIN {X 0,Y 98.279,Z 814.872,A -85,B 0,C 180,E1 24790.743,E2 24790.743} C_VEL
LIN {X 0,Y 117.185,Z 801.117,A -85,B 0,C 180,E1 24806.837,E2 24806.837} C_VEL
LIN {X 0,Y 141.935,Z 781.609,A -85,B 0,C 180,E1 24817.976,E2 24817.976} C_VEL
LIN {X 0,Y 168.571,Z 756.529,A -85,B 0,C 180,E1 24825.327,E2 24825.327} C_VEL
LIN {X 0,Y 192.161,Z 729.059,A -85,B 0,C 180,E1 24829.78,E2 24829.78} C_VEL
LIN {X 0,Y 193.537,Z 720.328,A -85,B 0,C 180,E1 24834.371,E2 24834.371} C_VEL
LIN {X 0,Y 194.032,Z 708.32,A -85,B 0,C 180,E1 24843.306,E2 24843.306} C_VEL
LIN {X 0,Y 194.168,Z 703.408,A -85,B 0,C 180,E1 24848.902,E2 24848.902} C_VEL
LIN {X 0,Y 192.059,Z 702.928,A -85,B 0,C 180,E1 24858.274,E2 24858.274} C_VEL
LIN {X 0,Y 191.091,Z 705.706,A -85,B 0,C 180,E1 24865.694,E2 24865.694} C_VEL
LIN {X 0,Y 189.915,Z 711.693,A -85,B 0,C 180,E1 24872.719,E2 24872.719} C_VEL
LIN {X 0,Y 187.866,Z 721.748,A -85,B 0,C 180,E1 24880.572,E2 24880.572} C_VEL
LIN {X 0,Y 187.113,Z 724.62,A -85,B 0,C 180,E1 24882.333,E2 24882.333} C_VEL
LIN {X 0,Y 162.134,Z 752.123,A -85,B 0,C 180,E1 24887.863,E2 24887.863} C_VEL
LIN {X 0,Y 137.469,Z 773.945,A -85,B 0,C 180,E1 24895.76,E2 24895.76} C_VEL
LIN {X 0,Y 113.65,Z 791.547,A -85,B 0,C 180,E1 24908.143,E2 24908.143} C_VEL
LIN {X 0,Y 96.422,Z 803.258,A -85,B 0,C 180,E1 24925.505,E2 24925.505} C_VEL
LIN {X 0,Y 87.99,Z 809.408,A -85,B 0,C 180,E1 24944.527,E2 24944.527} C_VEL
LIN {X 0,Y 86.975,Z 811.776,A -85,B 0,C 180,E1 24961.357,E2 24961.357} C_VEL
LIN {X 0,Y 94.743,Z 811.462,A -85,B 0,C 180,E1 24982.774,E2 24982.774} C_VEL
LIN {X 0,Y 114.877,Z 805.924,A -85,B 0,C 180,E1 25002.702,E2 25002.702} C_VEL
LIN {X 0,Y 122.83,Z 802.842,A -85,B 0,C 180,E1 25010.101,E2 25010.101} C_VEL
LIN {X 0,Y 132.379,Z 799.036,A -85,B 0,C 180,E1 25016.485,E2 25016.485} C_VEL
LIN {X 0,Y 164.598,Z 784.014,A -85,B 0,C 180,E1 25025.303,E2 25025.303} C_VEL
LIN {X 0,Y 186.833,Z 770.755,A -85,B 0,C 180,E1 25029.333,E2 25029.333} C_VEL
LIN {X 0,Y 183.942,Z 772.921,A -85,B 0,C 180,E1 25030.137,E2 25030.137} C_VEL
LIN {X 0,Y 149.65,Z 794.297,A -85,B 0,C 180,E1 25036.691,E2 25036.691} C_VEL
LIN {X 0,Y 115.841,Z 810.982,A -85,B 0,C 180,E1 25048.454,E2 25048.454} C_VEL
LIN {X 0,Y 90.375,Z 821.477,A -85,B 0,C 180,E1 25068.105,E2 25068.105} C_VEL
LIN {X 0,Y 80.253,Z 825.609,A -85,B 0,C 180,E1 25090.305,E2 25090.305} C_VEL
LIN {X 0,Y 79.885,Z 826.027,A -85,B 0,C 180,E1 25110.008,E2 25110.008} C_VEL
LIN {X 0,Y 81.023,Z 822.486,A -85,B 0,C 180,E1 25131.878,E2 25131.878} C_VEL
LIN {X 0,Y 92.2,Z 813.767,A -85,B 0,C 180,E1 25154.084,E2 25154.084} C_VEL
LIN {X 0,Y 115.586,Z 797.912,A -85,B 0,C 180,E1 25171.803,E2 25171.803} C_VEL
LIN {X 0,Y 142.601,Z 777.017,A -85,B 0,C 180,E1 25182.262,E2 25182.262} C_VEL
LIN {X 0,Y 169.337,Z 751.724,A -85,B 0,C 180,E1 25188.611,E2 25188.611} C_VEL
LIN {X 0,Y 187.285,Z 730.816,A -85,B 0,C 180,E1 25191.878,E2 25191.878} C_VEL
LIN {X 0,Y 188.542,Z 720.191,A -85,B 0,C 180,E1 25198.816,E2 25198.816} C_VEL
LIN {X 0,Y 189.265,Z 711.397,A -85,B 0,C 180,E1 25206.829,E2 25206.829} C_VEL
LIN {X 0,Y 189.338,Z 709.693,A -85,B 0,C 180,E1 25209.131,E2 25209.131} C_VEL
LIN {X 0,Y 187.233,Z 709.409,A -85,B 0,C 180,E1 25218.762,E2 25218.762} C_VEL
LIN {X 0,Y 185.956,Z 712.793,A -85,B 0,C 180,E1 25226.786,E2 25226.786} C_VEL
LIN {X 0,Y 184.534,Z 718.466,A -85,B 0,C 180,E1 25233.133,E2 25233.133} C_VEL
LIN {X 0,Y 181.842,Z 727.915,A -85,B 0,C 180,E1 25240.477,E2 25240.477} C_VEL
LIN {X 0,Y 157.564,Z 753.574,A -85,B 0,C 180,E1 25245.588,E2 25245.588} C_VEL
LIN {X 0,Y 131.599,Z 775.54,A -85,B 0,C 180,E1 25253.503,E2 25253.503} C_VEL
LIN {X 0,Y 106.207,Z 793.263,A -85,B 0,C 180,E1 25266.523,E2 25266.523} C_VEL
LIN {X 0,Y 88.216,Z 804.625,A -85,B 0,C 180,E1 25285.086,E2 25285.086} C_VEL
LIN {X 0,Y 79.291,Z 810.863,A -85,B 0,C 180,E1 25308.24,E2 25308.24} C_VEL
LIN {X 0,Y 83.117,Z 812.868,A -85,B 0,C 180,E1 25336.558,E2 25336.558} C_VEL
LIN {X 0,Y 100.647,Z 809.563,A -85,B 0,C 180,E1 25359.245,E2 25359.245} C_VEL
LIN {X 0,Y 129.361,Z 800.201,A -85,B 0,C 180,E1 25375.354,E2 25375.354} C_VEL
LIN {X 0,Y 132.379,Z 799.036,A -85,B 0,C 180,E1 25376.485,E2 25376.485} C_VEL
LIN {X 0,Y 143.26,Z 794.544,A -85,B 0,C 180,E1 25381.904,E2 25381.904} C_VEL
LIN {X 0,Y 154.981,Z 789.178,A -85,B 0,C 180,E1 25386.46,E2 25386.46} C_VEL
LIN {X 0,Y 168.027,Z 782.465,A -85,B 0,C 180,E1 25388.953,E2 25388.953} C_VEL
LIN {X 0,Y 168.385,Z 782.415,A -85,B 0,C 180,E1 25389.696,E2 25389.696} C_VEL
LIN {X 0,Y 133.271,Z 801.384,A -85,B 0,C 180,E1 25397.212,E2 25397.212} C_VEL
LIN {X 0,Y 98.904,Z 815.83,A -85,B 0,C 180,E1 25411.883,E2 25411.883} C_VEL
LIN {X 0,Y 77.7,Z 823.247,A -85,B 0,C 180,E1 25434.374,E2 25434.374} C_VEL
LIN {X 0,Y 71.385,Z 825.393,A -85,B 0,C 180,E1 25457.805,E2 25457.805} C_VEL
LIN {X 0,Y 71.972,Z 825.234,A -85,B 0,C 180,E1 25470.009,E2 25470.009} C_VEL
LIN {X 0,Y 73.579,Z 821.565,A -85,B 0,C 180,E1 25494.225,E2 25494.225} C_VEL
LIN {X 0,Y 88.624,Z 811.394,A -85,B 0,C 180,E1 25520.027,E2 25520.027} C_VEL
LIN {X 0,Y 114.052,Z 795,A -85,B 0,C 180,E1 25536.551,E2 25536.551} C_VEL
LIN {X 0,Y 141.934,Z 773.89,A -85,B 0,C 180,E1 25545.9,E2 25545.9} C_VEL
LIN {X 0,Y 168.946,Z 748.479,A -85,B 0,C 180,E1 25551.569,E2 25551.569} C_VEL
LIN {X 0,Y 181.874,Z 733.868,A -85,B 0,C 180,E1 25553.71,E2 25553.71} C_VEL
LIN {X 0,Y 183.476,Z 723.558,A -85,B 0,C 180,E1 25561.139,E2 25561.139} C_VEL
LIN {X 0,Y 184.226,Z 717.555,A -85,B 0,C 180,E1 25567.017,E2 25567.017} C_VEL
LIN {X 0,Y 184.07,Z 715.748,A -85,B 0,C 180,E1 25570.319,E2 25570.319} C_VEL
LIN {X 0,Y 182.145,Z 715.825,A -85,B 0,C 180,E1 25579.306,E2 25579.306} C_VEL
LIN {X 0,Y 181.257,Z 717.734,A -85,B 0,C 180,E1 25584.549,E2 25584.549} C_VEL
LIN {X 0,Y 179.746,Z 722.254,A -85,B 0,C 180,E1 25590.828,E2 25590.828} C_VEL
LIN {X 0,Y 177.105,Z 730.211,A -85,B 0,C 180,E1 25597.895,E2 25597.895} C_VEL
LIN {X 0,Y 175.385,Z 732.641,A -85,B 0,C 180,E1 25598.736,E2 25598.736} C_VEL
LIN {X 0,Y 147.926,Z 759.745,A -85,B 0,C 180,E1 25604.426,E2 25604.426} C_VEL
LIN {X 0,Y 119.947,Z 781.31,A -85,B 0,C 180,E1 25613.297,E2 25613.297} C_VEL
LIN {X 0,Y 95.857,Z 796.626,A -85,B 0,C 180,E1 25626.816,E2 25626.816} C_VEL
LIN {X 0,Y 79.988,Z 805.913,A -85,B 0,C 180,E1 25644.579,E2 25644.579} C_VEL
LIN {X 0,Y 72.584,Z 810.527,A -85,B 0,C 180,E1 25661.99,E2 25661.99} C_VEL
LIN {X 0,Y 72.365,Z 813.485,A -85,B 0,C 180,E1 25688.713,E2 25688.713} C_VEL
LIN {X 0,Y 84.785,Z 812.548,A -85,B 0,C 180,E1 25712.845,E2 25712.845} C_VEL
LIN {X 0,Y 107.122,Z 807.421,A -85,B 0,C 180,E1 25730.393,E2 25730.393} C_VEL
LIN {X 0,Y 139.749,Z 795.994,A -85,B 0,C 180,E1 25742.82,E2 25742.82} C_VEL
LIN {X 0,Y 154.981,Z 789.178,A -85,B 0,C 180,E1 25746.46,E2 25746.46} C_VEL
LIN {X 0,Y 154.445,Z 789.669,A -85,B 0,C 180,E1 25747.971,E2 25747.971} C_VEL
LIN {X 0,Y 144.978,Z 794.701,A -85,B 0,C 180,E1 25750.651,E2 25750.651} C_VEL
LIN {X 0,Y 138.331,Z 797.919,A -85,B 0,C 180,E1 25752.106,E2 25752.106} C_VEL
LIN {X 0,Y 102.828,Z 812.587,A -85,B 0,C 180,E1 25763.496,E2 25763.496} C_VEL
LIN {X 0,Y 76.096,Z 821.178,A -85,B 0,C 180,E1 25783.401,E2 25783.401} C_VEL
LIN {X 0,Y 64.228,Z 824.495,A -85,B 0,C 180,E1 25810.307,E2 25810.307} C_VEL
LIN {X 0,Y 64.044,Z 824.435,A -85,B 0,C 180,E1 25830.01,E2 25830.01} C_VEL
LIN {X 0,Y 66.29,Z 820.641,A -85,B 0,C 180,E1 25857.094,E2 25857.094} C_VEL
LIN {X 0,Y 83.575,Z 810.182,A -85,B 0,C 180,E1 25884.355,E2 25884.355} C_VEL
LIN {X 0,Y 110.348,Z 793.94,A -85,B 0,C 180,E1 25900.234,E2 25900.234} C_VEL
LIN {X 0,Y 138.457,Z 773.48,A -85,B 0,C 180,E1 25908.804,E2 25908.804} C_VEL
LIN {X 0,Y 165.04,Z 749.236,A -85,B 0,C 180,E1 25913.937,E2 25913.937} C_VEL
LIN {X 0,Y 176.477,Z 736.871,A -85,B 0,C 180,E1 25915.669,E2 25915.669} C_VEL
LIN {X 0,Y 178.438,Z 726.953,A -85,B 0,C 180,E1 25923.595,E2 25923.595} C_VEL
LIN {X 0,Y 179.274,Z 721.937,A -85,B 0,C 180,E1 25929.649,E2 25929.649} C_VEL
LIN {X 0,Y 178.02,Z 721.465,A -85,B 0,C 180,E1 25934.687,E2 25934.687} C_VEL
LIN {X 0,Y 176.433,Z 722.832,A -85,B 0,C 180,E1 25942.217,E2 25942.217} C_VEL
LIN {X 0,Y 174.478,Z 727.716,A -85,B 0,C 180,E1 25950.125,E2 25950.125} C_VEL
LIN {X 0,Y 171.422,Z 734.773,A -85,B 0,C 180,E1 25956.504,E2 25956.504} C_VEL
LIN {X 0,Y 144.419,Z 760.52,A -85,B 0,C 180,E1 25961.668,E2 25961.668} C_VEL
LIN {X 0,Y 115.142,Z 782.241,A -85,B 0,C 180,E1 25970.283,E2 25970.283} C_VEL
LIN {X 0,Y 88.463,Z 798.185,A -85,B 0,C 180,E1 25984.749,E2 25984.749} C_VEL
LIN {X 0,Y 71.707,Z 807.151,A -85,B 0,C 180,E1 26003.951,E2 26003.951} C_VEL
LIN {X 0,Y 63.362,Z 812.25,A -85,B 0,C 180,E1 26028.117,E2 26028.117} C_VEL
LIN {X 0,Y 66.954,Z 814.35,A -85,B 0,C 180,E1 26057.615,E2 26057.615} C_VEL
LIN {X 0,Y 85.468,Z 812.343,A -85,B 0,C 180,E1 26082.849,E2 26082.849} C_VEL
LIN {X 0,Y 113.448,Z 805.557,A -85,B 0,C 180,E1 26098.659,E2 26098.659} C_VEL
LIN {X 0,Y 147.93,Z 792.837,A -85,B 0,C 180,E1 26108.295,E2 26108.295} C_VEL
LIN {X 0,Y 152.691,Z 790.77,A -85,B 0,C 180,E1 26109.221,E2 26109.221} C_VEL
LIN {X 0,Y 138.331,Z 797.919,A -85,B 0,C 180,E1 26112.106,E2 26112.106} C_VEL
LIN {X 0,Y 132.988,Z 800.011,A -85,B 0,C 180,E1 26111.674,E2 26111.674} C_VEL
LIN {X 0,Y 120.664,Z 803.638,A -85,B 0,C 180,E1 26105.574,E2 26105.574} C_VEL
LIN {X 0,Y 91.032,Z 811.36,A -85,B 0,C 180,E1 26093.977,E2 26093.977} C_VEL
LIN {X 0,Y 66.754,Z 814.887,A -85,B 0,C 180,E1 26073.248,E2 26073.248} C_VEL
LIN {X 0,Y 55.388,Z 814.358,A -85,B 0,C 180,E1 26043.003,E2 26043.003} C_VEL
LIN {X 0,Y 60.221,Z 810.01,A -85,B 0,C 180,E1 26009.877,E2 26009.877} C_VEL
LIN {X 0,Y 78.67,Z 800.983,A -85,B 0,C 180,E1 25984.423,E2 25984.423} C_VEL
LIN {X 0,Y 104.349,Z 787.045,A -85,B 0,C 180,E1 25969.393,E2 25969.393} C_VEL
